// TIA Portal project "EB23" (V15)
// Maquina Raumak 23

(* hardware
DEVICE "S7-1200 station_1"  S7-1200 Station
   slot 0: "Rack_0"  S7-1200 Rack  Rack  V1.0
   slot 1: "PLC_1"  CPU 1214C DC/DC/Rly  6ES7 214-1HG40-0XB0  V4.2
   slot 2: "DI 16x24VDC_1"  6ES7 221-1BH32-0XB0  V2.0
   slot 3: "DQ 16x24VDC_1"  SM 1222 DQ16 x 24VDC  6ES7 222-1BH32-0XB0  V2.0
DEVICE "HMI_1"  KTP700 Basic PN
   slot 0: "HMI_1"  KTP700 Basic PN  6AV2 123-2GB03-0AX0  15.0.0.0
   slot 1: "HMI_RT_1"  KTP700 Basic PN  6AV2 123-2GB03-0AX0  15.0.0.0
   slot 5: "HMI_1.IE_CP_1"  PROFINET Interface  15.0.0.0
      slot 1: "PROFINET Interface_1"  PROFINET Interface
         slot 1: "Port_1"  Port
*)

// ===== PLC "PLC_1"  CPU 1214C DC/DC/Rly =====

VAR_GLOBAL   // PLC tag table "Default tag table"
   "System_Byte" AT %MB1 : Byte;
   "FirstScan" AT %M1.0 : Bool;
   "DiagStatusUpdate" AT %M1.1 : Bool;
   "AlwaysTRUE" AT %M1.2 : Bool;
   "AlwaysFALSE" AT %M1.3 : Bool;
   "Clock_Byte" AT %MB0 : Byte;
   "Clock_10Hz" AT %M0.0 : Bool;
   "Clock_5Hz" AT %M0.1 : Bool;
   "Clock_2.5Hz" AT %M0.2 : Bool;
   "Clock_2Hz" AT %M0.3 : Bool;
   "Clock_1.25Hz" AT %M0.4 : Bool;
   "Clock_1Hz" AT %M0.5 : Bool;
   "Clock_0.625Hz" AT %M0.6 : Bool;
   "Clock_0.5Hz" AT %M0.7 : Bool;
   "E_stop_bit" AT %M10.0 : Bool;
   "F_Blender_bit" AT %M10.1 : Bool;
   "F_Collector_bit" AT %M10.2 : Bool;
   "F_puller_bit" AT %M10.3 : Bool;
   "F_servo_bit" AT %M10.4 : Bool;
   "F_unwinder_bit" AT %M10.5 : Bool;
   "Global_Alarm" AT %M10.6 : Bool;
   "Doser_pulse" AT %I0.0 : Bool;   // HSC in
   "Stop" AT %I0.2 : Bool;   // Stops machine
   "Start" AT %I0.3 : Bool;   // Start machine
   "F_Collector" AT %I0.4 : Bool;   // Collector band termic fuse
   "S_Horizontalsealer" AT %I0.5 : Bool;   // Sensor Horizontal Sealer
   "S_Photocell" AT %I0.6 : Bool;   // Photocell sensor
   "F_Unwinder" AT %I0.7 : Bool;   // Unwinder Motor thermic fuse
   "S_Reedlvl" AT %I1.0 : Bool;   // level Switch
   "F_Servo" AT %I1.1 : Bool;   // Servo motor termic fuse
   "F_Puller" AT %I1.2 : Bool;   // Puller motor termic fuse
   "S_OpenDoor" AT %I1.3 : Bool;   // Sensor Action Open Door
   "F_Blender" AT %I1.4 : Bool;   // Blender Motor thermic fuse
   "E_stop" AT %I1.5 : Bool;   // Emergency Stop
   "S_StuckCoil" AT %I8.0 : Bool;   // Sensor Stuck coil
   "S_UnwinderOn" AT %I8.1 : Bool;   // Sensor unwinder On
   "S_UnwinderOff" AT %I8.2 : Bool;   // Sensor unwinder Off
   "S_LooseCoil" AT %I8.3 : Bool;   // Sensor Loose Coil
   "S_knife" AT %I8.4 : Bool;   // Sensor Knife
   "Stop_remote" AT %I8.5 : Bool;   // Stop Remote
   "Dater_fault" AT %I8.6 : Bool;   // Dater Fault (Print)
   "Coder" AT %Q0.0 : Bool;   // Out Coder EV
   "Horizontal_sealer" AT %Q0.1 : Bool;   // Out Horizontal Sealer EV
   "Vertical_sealer" AT %Q0.2 : Bool;   // Out Vertical Sealer EV
   "Knife" AT %Q0.3 : Bool;   // Out Knife EV
   "Puller" AT %Q0.4 : Bool;   // Out Drive Puller
   "Pusher" AT %Q0.5 : Bool;   // Out Pusher EV
   "HorizontalHeater" AT %Q0.6 : Bool;   // Out KS Horizontal Heater
   "VerticalHeater" AT %Q0.7 : Bool;   // Out KS Vertical Heater
   "Feeder" AT %Q1.0 : Bool;   // Out Feeder EV
   "Doser" AT %Q1.1 : Bool;   // Out Servo Drive Doser
   "Unwinder" AT %Q12.0 : Bool;   // Out Unwinder motor
   "CollectorBelt" AT %Q12.1 : Bool;   // Out Collector Belt motor
   "Blender" AT %Q12.2 : Bool;   // Out Blender motor
   "En_io_doser" AT %Q12.3 : Bool;   // Out Enable and Reset Servo Drive Doser
   "dater" AT %Q12.4 : Bool;   // Out dater(Print)
   "Doser_pulse_bit" AT %M10.7 : Bool;
   "Stop_bit" AT %M11.0 : Bool;
   "Start_bit" AT %M11.1 : Bool;
   "S_Horizontalsealer_bit" AT %M11.2 : Bool;
   "S_Photocell_bit" AT %M11.3 : Bool;
   "S_Reedlvl_bit" AT %M11.4 : Bool;
   "S_OpenDoor_bit" AT %M11.5 : Bool;
   "S_StuckCoil_bit" AT %M11.7 : Bool;
   "S_UnwinderOn_bit" AT %M12.0 : Bool;
   "S_UnwinderOff_bit" AT %M12.1 : Bool;
   "S_LooseCoil_bit" AT %M12.2 : Bool;
   "S_knife_bit" AT %M12.3 : Bool;
   "Stop_remote_bit" AT %M12.4 : Bool;
   "Dater_fault_bit" AT %M12.5 : Bool;
   "Coder_bit" AT %M12.6 : Bool;
   "Horizontal_sealer_bit" AT %M12.7 : Bool;
   "Vertical_sealer_bit" AT %M13.0 : Bool;
   "Knife_bit" AT %M13.1 : Bool;
   "Puller_bit" AT %M13.2 : Bool;
   "Pusher_bit" AT %M13.3 : Bool;
   "HorizontalHeater_bit" AT %M13.4 : Bool;
   "VerticalHeater_bit" AT %M13.5 : Bool;
   "Feeder_bit" AT %M13.6 : Bool;
   "Doser_bit" AT %M13.7 : Bool;
   "Unwinder_bit" AT %M14.0 : Bool;
   "CollectorBelt_bit" AT %M14.1 : Bool;
   "Blender_bit" AT %M14.2 : Bool;
   "En_io_doser_bit" AT %M14.3 : Bool;
   "dater_bit" AT %M14.4 : Bool;
   "ONS0" AT %M14.5 : Bool;
   "Stop_machine" AT %M14.6 : Bool;
   "Run" AT %M14.7 : Bool;
   "En_opendoor" AT %M15.0 : Bool;
   "Stop_1" AT %M15.1 : Bool;
   "Stop_2" AT %M15.2 : Bool;
   "Stop_3" AT %M15.3 : Bool;
   "Stop_4" AT %M15.4 : Bool;
   "Stop_5" AT %M15.5 : Bool;
   "Stop_6" AT %M15.6 : Bool;
   "En_conectionHMI" AT %M15.7 : Bool;
   "Stage_1" AT %M16.0 : Bool;   // Ingreso a Etapa
   "Stage_2" AT %M16.1 : Bool;   // Sellado EV Vertical
   "Stage_3" AT %M16.2 : Bool;   // Sellado EV Horizontal
   "Stage_4" AT %M16.3 : Bool;   // Dater Print
   "Stage_5" AT %M16.4 : Bool;   // Maquina armada... lista a Dispensar
   "Stage_6" AT %M16.5 : Bool;   // Etapa de Confirmacion de sellado
   "T_puller_run" AT %MD17 : Time;
   "Stage_0" AT %M16.6 : Bool;   // Etapa de Reinicio
   "E_Manual_hmi" AT %M16.7 : Bool;
   "E_Manual" AT %M21.0 : Bool;
   "En_Verticalsealer_hmi" AT %M21.1 : Bool;
   "TestVerticalsealer_hmi" AT %M21.2 : Bool;
   "En_Horizontalsealer_hmi" AT %M21.3 : Bool;
   "Testhorizontalsealer_hmi" AT %M21.4 : Bool;
   "En_dater_hmi" AT %M21.5 : Bool;
   "Testdater_hmi" AT %M21.6 : Bool;
   "En_doser_hmi" AT %M21.7 : Bool;
   "En_knife_hmi" AT %M22.0 : Bool;
   "Tag_2" AT %M22.1 : Bool;
   "TestKnife_hmi" AT %M22.2 : Bool;
   "Stage_7" AT %M22.3 : Bool;   // Dosificar
   "Stage_8" AT %M22.4 : Bool;   // Corte cuchillo Ristra
   "Stage_9_1" AT %M22.5 : Bool;
   "ONS2" AT %M22.6 : Bool;
   "Testdoser_hmi" AT %M22.7 : Bool;
   "Stage_9_2" AT %M23.0 : Bool;
   "En_colector_hmi" AT %M23.1 : Bool;
   "TestCollector_hmi" AT %M23.2 : Bool;
   "En_Feeder_hmi" AT %M23.3 : Bool;
   "Stage_Feed_1" AT %M23.4 : Bool;
   "Stage_Blender_1" AT %M23.5 : Bool;
   "TestFeeder_hmi" AT %M23.6 : Bool;
   "En_blender_hmi" AT %M23.7 : Bool;
   "TestBlender_hmi" AT %M24.0 : Bool;
   "En_pusher_hmi" AT %M24.1 : Bool;
   "En_cleaning_hmi" AT %M24.2 : Bool;
   "Stage_CleaningMachine" AT %M24.3 : Bool;
   "Stage_Pusher" AT %M24.4 : Bool;
   "TestPusher_hmi" AT %M24.5 : Bool;
   "En_horizontalheater_hmi" AT %M24.6 : Bool;
   "En_verticalheater_hmi" AT %M24.7 : Bool;
   "Stage_9_0" AT %M25.0 : Bool;
   "Stage_Feed_0" AT %M25.1 : Bool;
   "Stage_Unw_0" AT %M25.2 : Bool;
   "Stage_Unw_1" AT %M25.3 : Bool;
   "En_puller_hmi" AT %M25.4 : Bool;
   "ONS5" AT %M25.5 : Bool;
   "TestUnwinder_hmi" AT %M25.6 : Bool;
   "Stage_Puller_1" AT %M25.7 : Bool;
   "Tag_3" AT %M26.0 : Bool;
   "Et_puller" AT %MD27 : Time;
   "U_Coder_bit" AT %M31.0 : Bool;
   "TestPuller_hmi" AT %M31.1 : Bool;
   "Stage_Photo_1" AT %M31.2 : Bool;
   "ONS7" AT %M31.3 : Bool;
   "Stage_Photo_0" AT %M31.4 : Bool;
   "ONS8" AT %M31.5 : Bool;
   "reset_ppm" AT %M31.6 : Bool;
   "CV_ppm" AT %MW32 : Int;
   "ONS10" AT %M34.0 : Bool;
   "PPM" AT %MW36 : Int;
   "Total_vertical_sealer" AT %MD38 : Time;
   "High_Sealer" AT %MD42 : Time;
   "stimate_ppm" AT %MD46 : DInt;
   "ret_val_RD_LOC" AT %MW50 : Int;
   "ret_val_RD_SYS" AT %MW52 : Int;
   "ret_val_WR_SYS" AT %MW54 : Int;
   "ONS12" AT %M56.0 : Bool;
   "write_time" AT %M56.1 : Bool;
   "Stage_Blender_0" AT %M56.2 : Bool;
END_VAR

DATA_BLOCK "DB_Alarms"   // DB1
{ S7_Optimized_Access := 'FALSE' }
VERSION : 0.1
   VAR
      Alarms_active : Bool;
      E_stop_alm : Bool;
      Colector_alm : Bool;
      Puller_alm : Bool;
      "Unwinder-alm" : Bool;
      Servo_alm : Bool;
      Blender_alm : Bool;
      Open_door : Bool;
      Remote_stop : Bool;
      No_product : Bool;
      Blocked_jaws : Bool;
      Unwinder_loose : Bool;
      Unwinder_stuck : Bool;
      Stop_photocell : Bool;
      Coder_alm : Bool;
      Feed_alm : Bool;
   END_VAR
BEGIN
END_DATA_BLOCK

DATA_BLOCK "Init_Var"   // DB2
{ S7_Optimized_Access := 'TRUE' }
VERSION : 0.1
   VAR RETAIN
      Pt_cleaning : Time;
      Pt_coder : Time;
      Pt_collector : Time;
      Pt_collector_cut : Time;
      Pt_delay_doser : Time;
      Pt_delay_vert : Time;
      Pt_feeder : Time;
      Pt_horizontalsealer : Time;
      Pt_knife : Time;
      Pt_photocell : Time;
      Pt_preheat : Time;
      Pt_Puller : Time;
      Pt_pulses : Time;
      Pt_verticalsealer : Time;
      N_cycles : Int;
   END_VAR
BEGIN
END_DATA_BLOCK

DATA_BLOCK "DB_Time"   // DB22
{ S7_Optimized_Access := 'TRUE' }
VERSION : 0.1
   VAR
      time_local_READ : DTL;
      time_system_READ : DTL;
      time_system_WRITE : DTL;
   END_VAR
BEGIN
END_DATA_BLOCK

DATA_BLOCK "db_time_sync"   // DB22
{ S7_Optimized_Access := 'TRUE' }
VERSION : 0.1
   VAR
      time_local_READ : DTL;
      time_system_READ : DTL;
      time_system_WRITE : DTL;
   END_VAR
BEGIN
END_DATA_BLOCK

// folder: System blocks/Program resources

DATA_BLOCK "T_horizontal_stop"   // DB3
{ S7_Optimized_Access := 'TRUE' }
AUTHOR : Simatic
FAMILY : IEC
NAME : IEC_TMR
VERSION : 1.0
// stored: InstanceOfName IEC_TIMER
"IEC_TIMER"
BEGIN
END_DATA_BLOCK

DATA_BLOCK "T_delay_vert"   // DB4
{ S7_Optimized_Access := 'TRUE' }
AUTHOR : Simatic
FAMILY : IEC
NAME : IEC_TMR
VERSION : 1.0
// stored: InstanceOfName IEC_TIMER
"IEC_TIMER"
BEGIN
END_DATA_BLOCK

DATA_BLOCK "T_VerticalS"   // DB5
{ S7_Optimized_Access := 'TRUE' }
AUTHOR : Simatic
FAMILY : IEC
NAME : IEC_TMR
VERSION : 1.0
// stored: InstanceOfName IEC_TIMER
"IEC_TIMER"
BEGIN
END_DATA_BLOCK

DATA_BLOCK "T_HorizontalSealer"   // DB6
{ S7_Optimized_Access := 'TRUE' }
AUTHOR : Simatic
FAMILY : IEC
NAME : IEC_TMR
VERSION : 1.0
// stored: InstanceOfName IEC_TIMER
"IEC_TIMER"
BEGIN
END_DATA_BLOCK

DATA_BLOCK "Packages_Knife"   // DB7
{ S7_Optimized_Access := 'TRUE' }
AUTHOR : Simatic
FAMILY : IEC
NAME : CNTR
VERSION : 1.0
// stored: InstanceOfName IEC_COUNTER
"IEC_COUNTER"
BEGIN
END_DATA_BLOCK

DATA_BLOCK "T_Knife"   // DB8
{ S7_Optimized_Access := 'TRUE' }
AUTHOR : Simatic
FAMILY : IEC
NAME : IEC_TMR
VERSION : 1.0
// stored: InstanceOfName IEC_TIMER
"IEC_TIMER"
BEGIN
END_DATA_BLOCK

DATA_BLOCK "T_DelayDoser"   // DB9
{ S7_Optimized_Access := 'TRUE' }
AUTHOR : Simatic
FAMILY : IEC
NAME : IEC_TMR
VERSION : 1.0
// stored: InstanceOfName IEC_TIMER
"IEC_TIMER"
BEGIN
END_DATA_BLOCK

DATA_BLOCK "T_PulseDoser"   // DB10
{ S7_Optimized_Access := 'TRUE' }
AUTHOR : Simatic
FAMILY : IEC
NAME : IEC_TMR
VERSION : 1.0
// stored: InstanceOfName IEC_TIMER
"IEC_TIMER"
BEGIN
END_DATA_BLOCK

DATA_BLOCK "T_CollectorCut"   // DB11
{ S7_Optimized_Access := 'TRUE' }
AUTHOR : Simatic
FAMILY : IEC
NAME : IEC_TMR
VERSION : 1.0
// stored: InstanceOfName IEC_TIMER
"IEC_TIMER"
BEGIN
END_DATA_BLOCK

DATA_BLOCK "T_Collector"   // DB12
{ S7_Optimized_Access := 'TRUE' }
AUTHOR : Simatic
FAMILY : IEC
NAME : IEC_TMR
VERSION : 1.0
// stored: InstanceOfName IEC_TIMER
"IEC_TIMER"
BEGIN
END_DATA_BLOCK

DATA_BLOCK "Cnt_LevelFeeder"   // DB13
{ S7_Optimized_Access := 'TRUE' }
AUTHOR : Simatic
FAMILY : IEC
NAME : CNTR
VERSION : 1.0
// stored: InstanceOfName IEC_COUNTER
"IEC_COUNTER"
BEGIN
END_DATA_BLOCK

DATA_BLOCK "T_Feeder"   // DB14
{ S7_Optimized_Access := 'TRUE' }
AUTHOR : Simatic
FAMILY : IEC
NAME : IEC_TMR
VERSION : 1.0
// stored: InstanceOfName IEC_TIMER
"IEC_TIMER"
BEGIN
END_DATA_BLOCK

DATA_BLOCK "T_CleanMachine"   // DB15
{ S7_Optimized_Access := 'TRUE' }
AUTHOR : Simatic
FAMILY : IEC
NAME : IEC_TMR
VERSION : 1.0
// stored: InstanceOfName IEC_TIMER
"IEC_TIMER"
BEGIN
END_DATA_BLOCK

DATA_BLOCK "T_Puller"   // DB16
{ S7_Optimized_Access := 'TRUE' }
AUTHOR : Simatic
FAMILY : IEC
NAME : IEC_TMR
VERSION : 1.0
// stored: InstanceOfName IEC_TIMER
"IEC_TIMER"
BEGIN
END_DATA_BLOCK

DATA_BLOCK "T_Puller_Running"   // DB17
{ S7_Optimized_Access := 'TRUE' }
AUTHOR : Simatic
FAMILY : IEC
NAME : IEC_TMR
VERSION : 1.0
// stored: InstanceOfName IEC_TIMER
"IEC_TIMER"
BEGIN
END_DATA_BLOCK

DATA_BLOCK "T_PhotoCell"   // DB18
{ S7_Optimized_Access := 'TRUE' }
AUTHOR : Simatic
FAMILY : IEC
NAME : IEC_TMR
VERSION : 1.0
// stored: InstanceOfName IEC_TIMER
"IEC_TIMER"
BEGIN
END_DATA_BLOCK

DATA_BLOCK "Packages_PPM"   // DB19
{ S7_Optimized_Access := 'TRUE' }
AUTHOR : Simatic
FAMILY : IEC
NAME : CNTR
VERSION : 1.0
// stored: InstanceOfName IEC_COUNTER
"IEC_COUNTER"
BEGIN
END_DATA_BLOCK

DATA_BLOCK "T_Delay_ppm"   // DB20
{ S7_Optimized_Access := 'TRUE' }
AUTHOR : Simatic
FAMILY : IEC
NAME : IEC_TMR
VERSION : 1.0
// stored: InstanceOfName IEC_TIMER
"IEC_TIMER"
BEGIN
END_DATA_BLOCK

DATA_BLOCK "T_ppm"   // DB21
{ S7_Optimized_Access := 'TRUE' }
AUTHOR : Simatic
FAMILY : IEC
NAME : IEC_TMR
VERSION : 1.0
// stored: InstanceOfName IEC_TIMER
"IEC_TIMER"
BEGIN
END_DATA_BLOCK

// folder: (top level)

ORGANIZATION_BLOCK "Main"   // OB1, LAD, ProgramCycle
TITLE = "Main Program Sweep (Cycle)"
{ S7_Optimized_Access := 'TRUE' }
VERSION : 0.1
   VAR_INPUT
      Initial_Call : Bool;   // Initial call of this OB
      Remanence : Bool;   // =True, if remanent data are available
   END_VAR
   VAR_TEMP   // added for the SCL form of the ladder/FBD networks
      _w1 : Bool;
   END_VAR
BEGIN

REGION Network 1
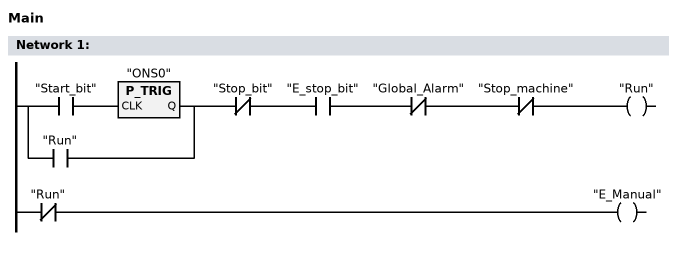
   RUNG wire#powerrail
      Contact( "Start_bit" )
      P_Trig( "ONS0" )
      wire#w1
      I_Contact( "Stop_bit" )
      Contact( "E_stop_bit" )
      I_Contact( "Global_Alarm" )
      I_Contact( "Stop_machine" )
      Coil( "Run" )
   END_RUNG
   RUNG wire#powerrail
      Contact( "Run" )
   END_RUNG wire#w1
   RUNG wire#powerrail
      I_Contact( "Run" )
      Coil( "E_Manual" )
   END_RUNG
   // the same network as SCL:
   #_w1 := "Start_bit" AND NOT "ONS0";   // rising edge
   "ONS0" := "Start_bit";
   "Run" := (#_w1 OR "Run") AND NOT "Stop_bit" AND "E_stop_bit" AND NOT "Global_Alarm" AND NOT "Stop_machine";
   "E_Manual" := NOT "Run";
END_REGION
END_ORGANIZATION_BLOCK

ORGANIZATION_BLOCK "Actions"   // OB123, LAD, ProgramCycle
TITLE = "Main Program Sweep (Cycle)"
{ S7_Optimized_Access := 'TRUE' }
VERSION : 0.1
   VAR_INPUT
      Initial_Call : Bool;   // Initial call of this OB
      Remanence : Bool;   // =True, if remanent data are available
   END_VAR
BEGIN

REGION Network 1: Peripherals EV
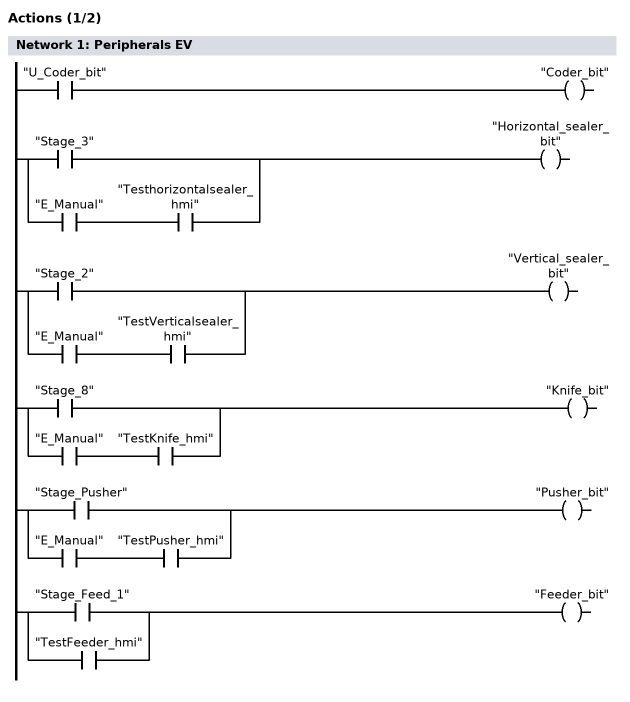
   RUNG wire#powerrail
      Contact( "U_Coder_bit" )
      Coil( "Coder_bit" )
   END_RUNG
   RUNG wire#powerrail
      Contact( "Stage_3" )
      wire#w1
      Coil( "Horizontal_sealer_bit" )
   END_RUNG
   RUNG wire#powerrail
      Contact( "E_Manual" )
      Contact( "Testhorizontalsealer_hmi" )
   END_RUNG wire#w1
   RUNG wire#powerrail
      Contact( "Stage_2" )
      wire#w2
      Coil( "Vertical_sealer_bit" )
   END_RUNG
   RUNG wire#powerrail
      Contact( "E_Manual" )
      Contact( "TestVerticalsealer_hmi" )
   END_RUNG wire#w2
   RUNG wire#powerrail
      Contact( "Stage_8" )
      wire#w3
      Coil( "Knife_bit" )
   END_RUNG
   RUNG wire#powerrail
      Contact( "E_Manual" )
      Contact( "TestKnife_hmi" )
   END_RUNG wire#w3
   RUNG wire#powerrail
      Contact( "Stage_Pusher" )
      wire#w4
      Coil( "Pusher_bit" )
   END_RUNG
   RUNG wire#powerrail
      Contact( "E_Manual" )
      Contact( "TestPusher_hmi" )
   END_RUNG wire#w4
   RUNG wire#powerrail
      Contact( "Stage_Feed_1" )
      wire#w5
      Coil( "Feeder_bit" )
   END_RUNG
   RUNG wire#powerrail
      Contact( "TestFeeder_hmi" )
   END_RUNG wire#w5
   // the same network as SCL:
   "Coder_bit" := "U_Coder_bit";
   "Horizontal_sealer_bit" := "Stage_3" OR ("E_Manual" AND "Testhorizontalsealer_hmi");
   "Vertical_sealer_bit" := "Stage_2" OR ("E_Manual" AND "TestVerticalsealer_hmi");
   "Knife_bit" := "Stage_8" OR ("E_Manual" AND "TestKnife_hmi");
   "Pusher_bit" := "Stage_Pusher" OR ("E_Manual" AND "TestPusher_hmi");
   "Feeder_bit" := "Stage_Feed_1" OR "TestFeeder_hmi";
END_REGION

REGION Network 2: Peripherals Motors
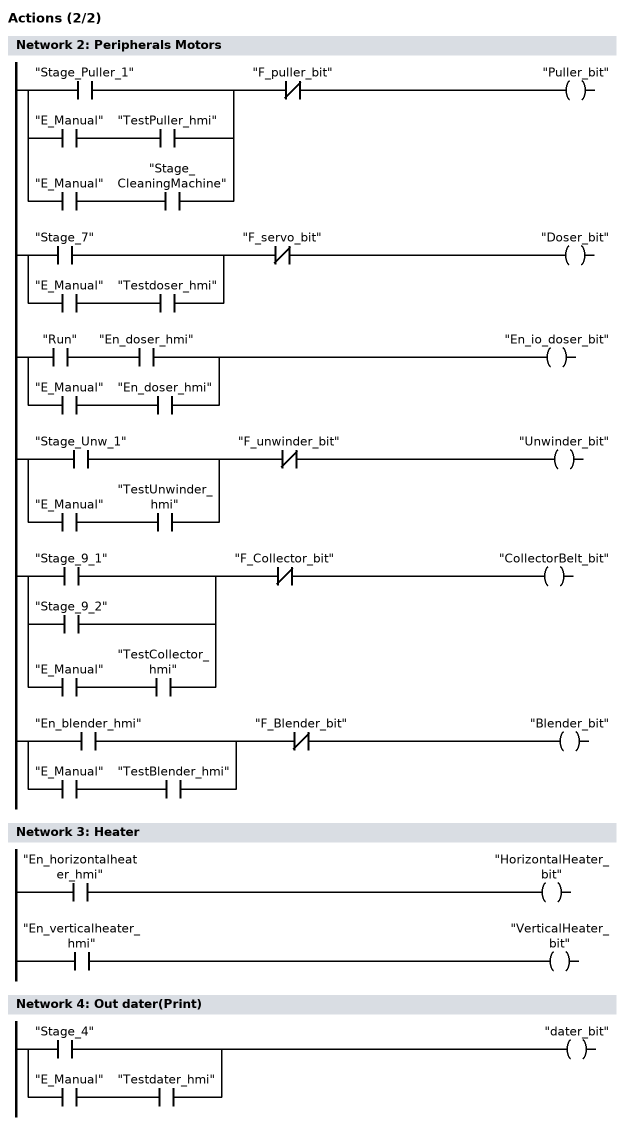
   RUNG wire#powerrail
      Contact( "Stage_Puller_1" )
      wire#w1
      I_Contact( "F_puller_bit" )
      Coil( "Puller_bit" )
   END_RUNG
   RUNG wire#powerrail
      Contact( "E_Manual" )
      Contact( "TestPuller_hmi" )
   END_RUNG wire#w1
   RUNG wire#powerrail
      Contact( "E_Manual" )
      Contact( "Stage_CleaningMachine" )
   END_RUNG wire#w1
   RUNG wire#powerrail
      Contact( "Stage_7" )
      wire#w2
      I_Contact( "F_servo_bit" )
      Coil( "Doser_bit" )
   END_RUNG
   RUNG wire#powerrail
      Contact( "E_Manual" )
      Contact( "Testdoser_hmi" )
   END_RUNG wire#w2
   RUNG wire#powerrail
      Contact( "Run" )
      Contact( "En_doser_hmi" )
      wire#w3
      Coil( "En_io_doser_bit" )
   END_RUNG
   RUNG wire#powerrail
      Contact( "E_Manual" )
      Contact( "En_doser_hmi" )
   END_RUNG wire#w3
   RUNG wire#powerrail
      Contact( "Stage_Unw_1" )
      wire#w4
      I_Contact( "F_unwinder_bit" )
      Coil( "Unwinder_bit" )
   END_RUNG
   RUNG wire#powerrail
      Contact( "E_Manual" )
      Contact( "TestUnwinder_hmi" )
   END_RUNG wire#w4
   RUNG wire#powerrail
      Contact( "Stage_9_1" )
      wire#w5
      I_Contact( "F_Collector_bit" )
      Coil( "CollectorBelt_bit" )
   END_RUNG
   RUNG wire#powerrail
      Contact( "Stage_9_2" )
   END_RUNG wire#w5
   RUNG wire#powerrail
      Contact( "E_Manual" )
      Contact( "TestCollector_hmi" )
   END_RUNG wire#w5
   RUNG wire#powerrail
      Contact( "En_blender_hmi" )
      wire#w6
      I_Contact( "F_Blender_bit" )
      Coil( "Blender_bit" )
   END_RUNG
   RUNG wire#powerrail
      Contact( "E_Manual" )
      Contact( "TestBlender_hmi" )
   END_RUNG wire#w6
   // the same network as SCL:
   "Puller_bit" := ("Stage_Puller_1" OR ("E_Manual" AND "TestPuller_hmi") OR ("E_Manual" AND "Stage_CleaningMachine")) AND NOT "F_puller_bit";
   "Doser_bit" := ("Stage_7" OR ("E_Manual" AND "Testdoser_hmi")) AND NOT "F_servo_bit";
   "En_io_doser_bit" := ("Run" AND "En_doser_hmi") OR ("E_Manual" AND "En_doser_hmi");
   "Unwinder_bit" := ("Stage_Unw_1" OR ("E_Manual" AND "TestUnwinder_hmi")) AND NOT "F_unwinder_bit";
   "CollectorBelt_bit" := ("Stage_9_1" OR "Stage_9_2" OR ("E_Manual" AND "TestCollector_hmi")) AND NOT "F_Collector_bit";
   "Blender_bit" := ("En_blender_hmi" OR ("E_Manual" AND "TestBlender_hmi")) AND NOT "F_Blender_bit";
END_REGION

REGION Network 3: Heater
   RUNG wire#powerrail
      Contact( "En_horizontalheater_hmi" )
      Coil( "HorizontalHeater_bit" )
   END_RUNG
   RUNG wire#powerrail
      Contact( "En_verticalheater_hmi" )
      Coil( "VerticalHeater_bit" )
   END_RUNG
   // the same network as SCL:
   "HorizontalHeater_bit" := "En_horizontalheater_hmi";
   "VerticalHeater_bit" := "En_verticalheater_hmi";
END_REGION

REGION Network 4: Out dater(Print)
   RUNG wire#powerrail
      Contact( "Stage_4" )
      wire#w1
      Coil( "dater_bit" )
   END_RUNG
   RUNG wire#powerrail
      Contact( "E_Manual" )
      Contact( "Testdater_hmi" )
   END_RUNG wire#w1
   // the same network as SCL:
   "dater_bit" := "Stage_4" OR ("E_Manual" AND "Testdater_hmi");
END_REGION
END_ORGANIZATION_BLOCK

ORGANIZATION_BLOCK "Alarms"   // OB124, LAD, ProgramCycle
TITLE = "Main Program Sweep (Cycle)"
{ S7_Optimized_Access := 'TRUE' }
VERSION : 0.1
   VAR_INPUT
      Initial_Call : Bool;   // Initial call of this OB
      Remanence : Bool;   // =True, if remanent data are available
   END_VAR
BEGIN

REGION Network 1: Global Alarm Fuses
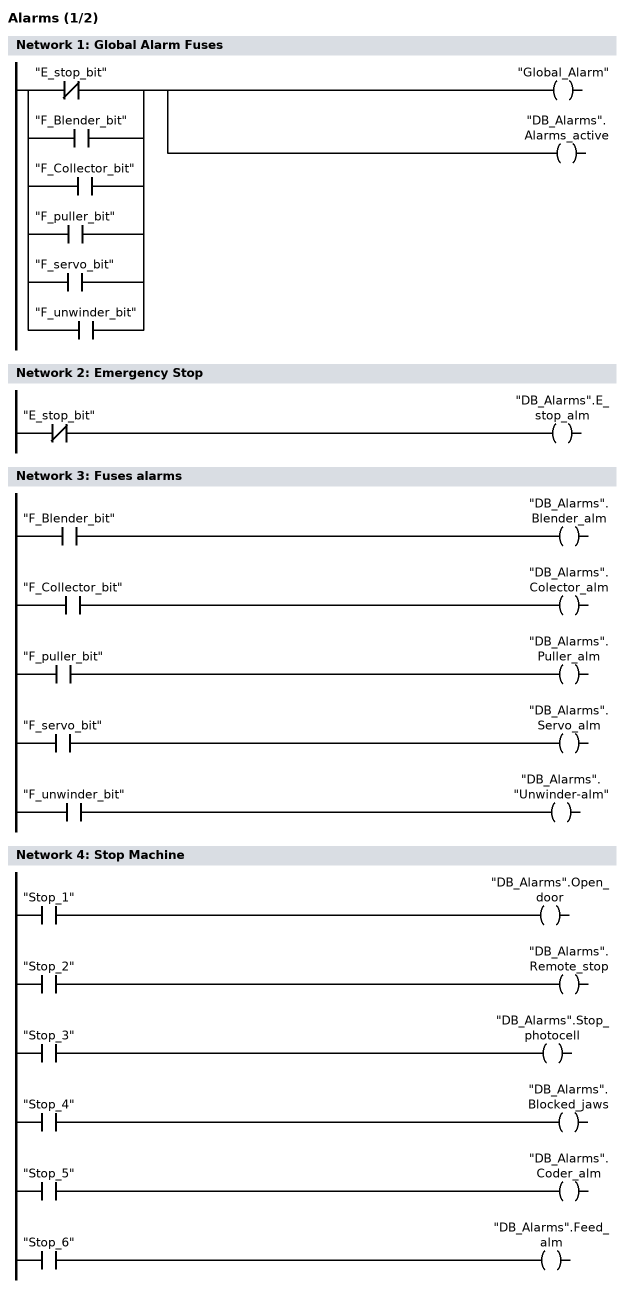
   RUNG wire#powerrail
      I_Contact( "E_stop_bit" )
      wire#w1
      Coil( "Global_Alarm" )
   END_RUNG
   RUNG wire#powerrail
      Contact( "F_Blender_bit" )
   END_RUNG wire#w1
   RUNG wire#powerrail
      Contact( "F_Collector_bit" )
   END_RUNG wire#w1
   RUNG wire#powerrail
      Contact( "F_puller_bit" )
   END_RUNG wire#w1
   RUNG wire#powerrail
      Contact( "F_servo_bit" )
   END_RUNG wire#w1
   RUNG wire#powerrail
      Contact( "F_unwinder_bit" )
   END_RUNG wire#w1
   RUNG wire#w1
      Coil( "DB_Alarms".Alarms_active )
   END_RUNG
   // the same network as SCL:
   "Global_Alarm" := NOT "E_stop_bit" OR "F_Blender_bit" OR "F_Collector_bit" OR "F_puller_bit" OR "F_servo_bit" OR "F_unwinder_bit";
   "DB_Alarms".Alarms_active := "Global_Alarm";
END_REGION

REGION Network 2: Emergency Stop
   RUNG wire#powerrail
      I_Contact( "E_stop_bit" )
      Coil( "DB_Alarms".E_stop_alm )
   END_RUNG
   // the same network as SCL:
   "DB_Alarms".E_stop_alm := NOT "E_stop_bit";
END_REGION

REGION Network 3: Fuses alarms
   RUNG wire#powerrail
      Contact( "F_Blender_bit" )
      Coil( "DB_Alarms".Blender_alm )
   END_RUNG
   RUNG wire#powerrail
      Contact( "F_Collector_bit" )
      Coil( "DB_Alarms".Colector_alm )
   END_RUNG
   RUNG wire#powerrail
      Contact( "F_puller_bit" )
      Coil( "DB_Alarms".Puller_alm )
   END_RUNG
   RUNG wire#powerrail
      Contact( "F_servo_bit" )
      Coil( "DB_Alarms".Servo_alm )
   END_RUNG
   RUNG wire#powerrail
      Contact( "F_unwinder_bit" )
      Coil( "DB_Alarms"."Unwinder-alm" )
   END_RUNG
   // the same network as SCL:
   "DB_Alarms".Blender_alm := "F_Blender_bit";
   "DB_Alarms".Colector_alm := "F_Collector_bit";
   "DB_Alarms".Puller_alm := "F_puller_bit";
   "DB_Alarms".Servo_alm := "F_servo_bit";
   "DB_Alarms"."Unwinder-alm" := "F_unwinder_bit";
END_REGION

REGION Network 4: Stop Machine
   RUNG wire#powerrail
      Contact( "Stop_1" )
      Coil( "DB_Alarms".Open_door )
   END_RUNG
   RUNG wire#powerrail
      Contact( "Stop_2" )
      Coil( "DB_Alarms".Remote_stop )
   END_RUNG
   RUNG wire#powerrail
      Contact( "Stop_3" )
      Coil( "DB_Alarms".Stop_photocell )
   END_RUNG
   RUNG wire#powerrail
      Contact( "Stop_4" )
      Coil( "DB_Alarms".Blocked_jaws )
   END_RUNG
   RUNG wire#powerrail
      Contact( "Stop_5" )
      Coil( "DB_Alarms".Coder_alm )
   END_RUNG
   RUNG wire#powerrail
      Contact( "Stop_6" )
      Coil( "DB_Alarms".Feed_alm )
   END_RUNG
   // the same network as SCL:
   "DB_Alarms".Open_door := "Stop_1";
   "DB_Alarms".Remote_stop := "Stop_2";
   "DB_Alarms".Stop_photocell := "Stop_3";
   "DB_Alarms".Blocked_jaws := "Stop_4";
   "DB_Alarms".Coder_alm := "Stop_5";
   "DB_Alarms".Feed_alm := "Stop_6";
END_REGION

REGION Network 5: Sensor Alarms
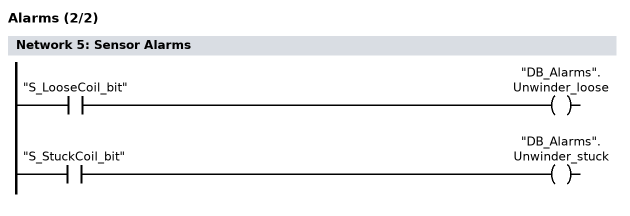
   RUNG wire#powerrail
      Contact( "S_LooseCoil_bit" )
      Coil( "DB_Alarms".Unwinder_loose )
   END_RUNG
   RUNG wire#powerrail
      Contact( "S_StuckCoil_bit" )
      Coil( "DB_Alarms".Unwinder_stuck )
   END_RUNG
   // the same network as SCL:
   "DB_Alarms".Unwinder_loose := "S_LooseCoil_bit";
   "DB_Alarms".Unwinder_stuck := "S_StuckCoil_bit";
END_REGION
END_ORGANIZATION_BLOCK

ORGANIZATION_BLOCK "Convertions"   // OB125, LAD, ProgramCycle
TITLE = "Main Program Sweep (Cycle)"
{ S7_Optimized_Access := 'TRUE' }
VERSION : 0.1
   VAR_INPUT
      Initial_Call : Bool;   // Initial call of this OB
      Remanence : Bool;   // =True, if remanent data are available
   END_VAR
   VAR_TEMP   // added for the SCL form of the ladder/FBD networks
      _w1 : Bool;
      _w2 : Bool;
      _w3 : Bool;
   END_VAR
BEGIN

REGION Network 2
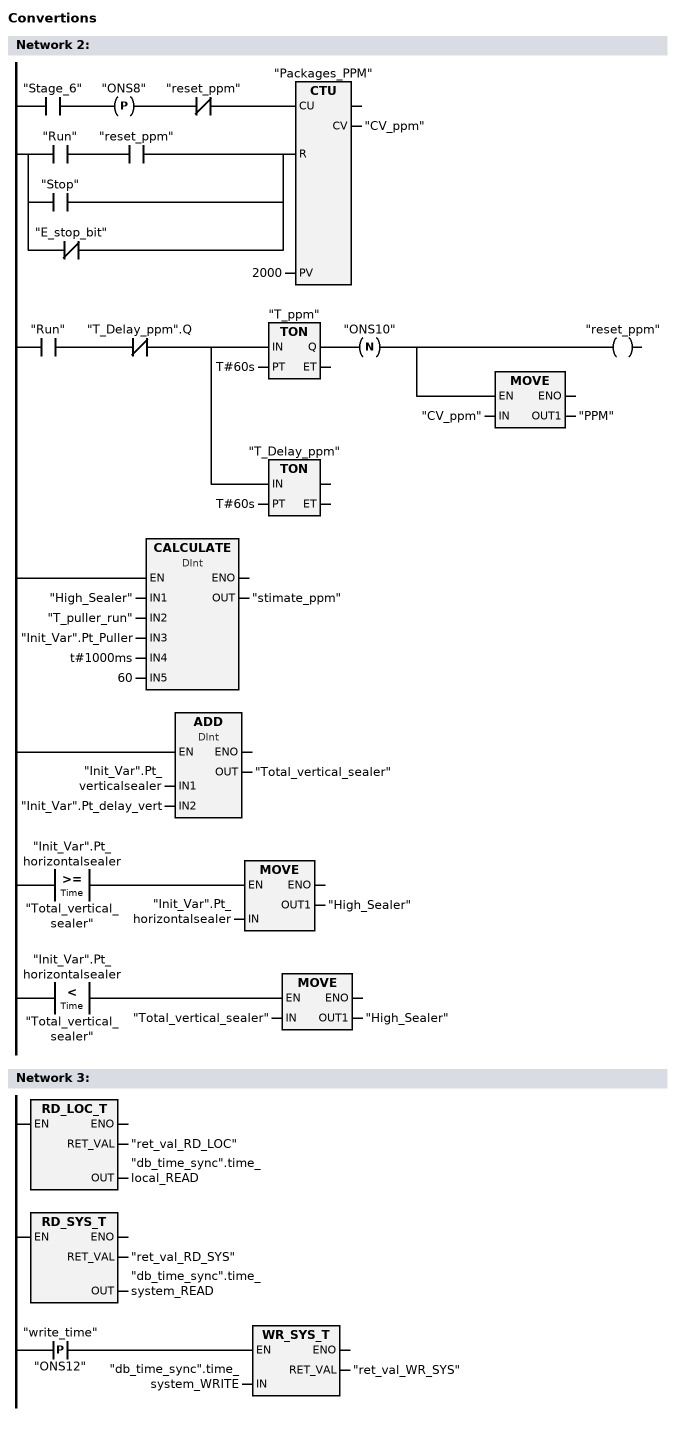
   #_w1 := "Stage_6" AND NOT "ONS8";   // rising edge
   "ONS8" := "Stage_6";
   "Packages_PPM".CTU(CU := #_w1 AND NOT "reset_ppm",
                      R := ("Run" AND "reset_ppm") OR "Stop" OR NOT "E_stop_bit",
                      PV := 2000,
                      CV => "CV_ppm");
   #_w2 := "Run" AND NOT "T_Delay_ppm".Q;
   "T_ppm".TON(IN := #_w2, PT := T#60s);
   #_w3 := NOT "T_ppm".Q AND "ONS10";   // falling edge
   "ONS10" := "T_ppm".Q;
   "reset_ppm" := #_w3;
   IF #_w3 THEN "PPM" := "CV_ppm"; END_IF;
   "T_Delay_ppm".TON(IN := #_w2, PT := T#60s);
   "stimate_ppm" := (t#1000ms*60)/("High_Sealer"+"T_puller_run"+"Init_Var".Pt_Puller);
   "Total_vertical_sealer" := "Init_Var".Pt_verticalsealer + "Init_Var".Pt_delay_vert;
   IF "Init_Var".Pt_horizontalsealer >= "Total_vertical_sealer" THEN
       "High_Sealer" := "Init_Var".Pt_horizontalsealer;
   END_IF;
   IF "Init_Var".Pt_horizontalsealer < "Total_vertical_sealer" THEN
       "High_Sealer" := "Total_vertical_sealer";
   END_IF;
END_REGION

REGION Network 3
   "ret_val_RD_LOC" := RD_LOC_T(OUT => "db_time_sync".time_local_READ);
   "ret_val_RD_SYS" := RD_SYS_T(OUT => "db_time_sync".time_system_READ);
   #_w1 := "write_time" AND NOT "ONS12";   // rising edge of "write_time"
   "ONS12" := "write_time";
   IF #_w1 THEN "ret_val_WR_SYS" := WR_SYS_T(IN := "db_time_sync".time_system_WRITE); END_IF;
END_REGION
END_ORGANIZATION_BLOCK

ORGANIZATION_BLOCK "Mirror_bit"   // OB126, LAD, ProgramCycle
TITLE = "Main Program Sweep (Cycle)"
{ S7_Optimized_Access := 'TRUE' }
VERSION : 0.1
   VAR_INPUT
      Initial_Call : Bool;   // Initial call of this OB
      Remanence : Bool;   // =True, if remanent data are available
   END_VAR
BEGIN

REGION Network 1: Inputs mirros Emergency
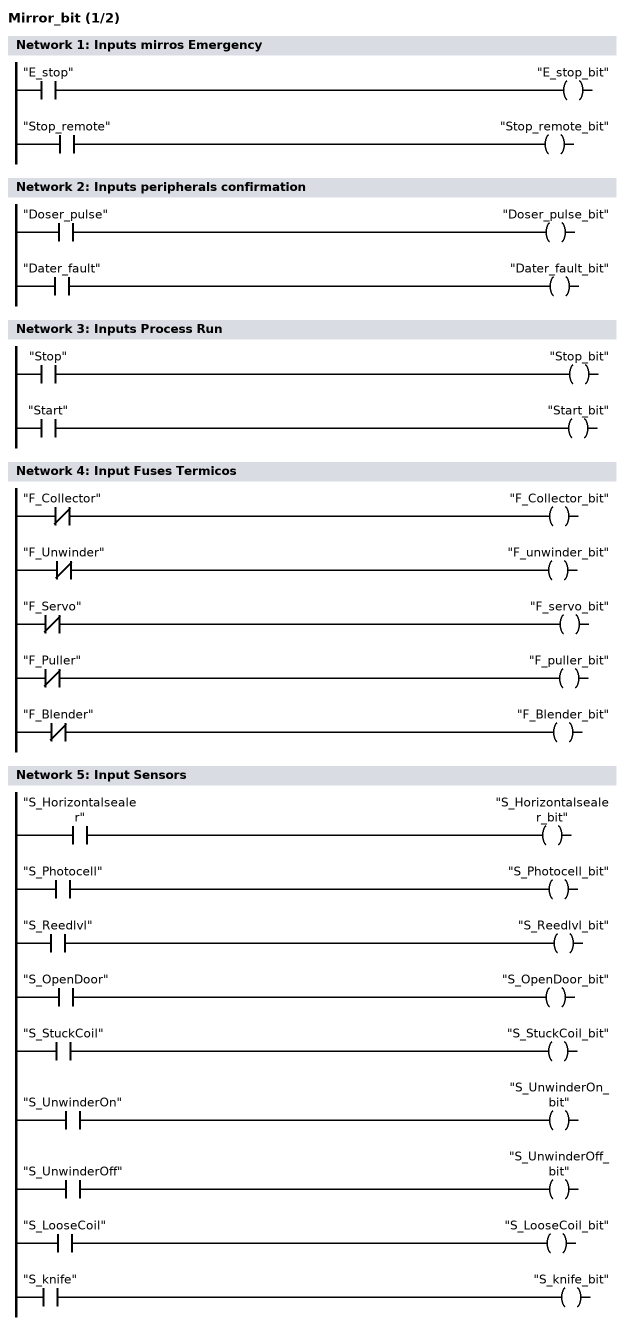
   RUNG wire#powerrail
      Contact( "E_stop" )
      Coil( "E_stop_bit" )
   END_RUNG
   RUNG wire#powerrail
      Contact( "Stop_remote" )
      Coil( "Stop_remote_bit" )
   END_RUNG
   // the same network as SCL:
   "E_stop_bit" := "E_stop";
   "Stop_remote_bit" := "Stop_remote";
END_REGION

REGION Network 2: Inputs peripherals confirmation
   RUNG wire#powerrail
      Contact( "Doser_pulse" )
      Coil( "Doser_pulse_bit" )
   END_RUNG
   RUNG wire#powerrail
      Contact( "Dater_fault" )
      Coil( "Dater_fault_bit" )
   END_RUNG
   // the same network as SCL:
   "Doser_pulse_bit" := "Doser_pulse";
   "Dater_fault_bit" := "Dater_fault";
END_REGION

REGION Network 3: Inputs Process Run
   RUNG wire#powerrail
      Contact( "Stop" )
      Coil( "Stop_bit" )
   END_RUNG
   RUNG wire#powerrail
      Contact( "Start" )
      Coil( "Start_bit" )
   END_RUNG
   // the same network as SCL:
   "Stop_bit" := "Stop";
   "Start_bit" := "Start";
END_REGION

REGION Network 4: Input Fuses Termicos
   RUNG wire#powerrail
      I_Contact( "F_Collector" )
      Coil( "F_Collector_bit" )
   END_RUNG
   RUNG wire#powerrail
      I_Contact( "F_Unwinder" )
      Coil( "F_unwinder_bit" )
   END_RUNG
   RUNG wire#powerrail
      I_Contact( "F_Servo" )
      Coil( "F_servo_bit" )
   END_RUNG
   RUNG wire#powerrail
      I_Contact( "F_Puller" )
      Coil( "F_puller_bit" )
   END_RUNG
   RUNG wire#powerrail
      I_Contact( "F_Blender" )
      Coil( "F_Blender_bit" )
   END_RUNG
   // the same network as SCL:
   "F_Collector_bit" := NOT "F_Collector";
   "F_unwinder_bit" := NOT "F_Unwinder";
   "F_servo_bit" := NOT "F_Servo";
   "F_puller_bit" := NOT "F_Puller";
   "F_Blender_bit" := NOT "F_Blender";
END_REGION

REGION Network 5: Input Sensors
   RUNG wire#powerrail
      Contact( "S_Horizontalsealer" )
      Coil( "S_Horizontalsealer_bit" )
   END_RUNG
   RUNG wire#powerrail
      Contact( "S_Photocell" )
      Coil( "S_Photocell_bit" )
   END_RUNG
   RUNG wire#powerrail
      Contact( "S_Reedlvl" )
      Coil( "S_Reedlvl_bit" )
   END_RUNG
   RUNG wire#powerrail
      Contact( "S_OpenDoor" )
      Coil( "S_OpenDoor_bit" )
   END_RUNG
   RUNG wire#powerrail
      Contact( "S_StuckCoil" )
      Coil( "S_StuckCoil_bit" )
   END_RUNG
   RUNG wire#powerrail
      Contact( "S_UnwinderOn" )
      Coil( "S_UnwinderOn_bit" )
   END_RUNG
   RUNG wire#powerrail
      Contact( "S_UnwinderOff" )
      Coil( "S_UnwinderOff_bit" )
   END_RUNG
   RUNG wire#powerrail
      Contact( "S_LooseCoil" )
      Coil( "S_LooseCoil_bit" )
   END_RUNG
   RUNG wire#powerrail
      Contact( "S_knife" )
      Coil( "S_knife_bit" )
   END_RUNG
   // the same network as SCL:
   "S_Horizontalsealer_bit" := "S_Horizontalsealer";
   "S_Photocell_bit" := "S_Photocell";
   "S_Reedlvl_bit" := "S_Reedlvl";
   "S_OpenDoor_bit" := "S_OpenDoor";
   "S_StuckCoil_bit" := "S_StuckCoil";
   "S_UnwinderOn_bit" := "S_UnwinderOn";
   "S_UnwinderOff_bit" := "S_UnwinderOff";
   "S_LooseCoil_bit" := "S_LooseCoil";
   "S_knife_bit" := "S_knife";
END_REGION

REGION Network 6: Peripherals EV
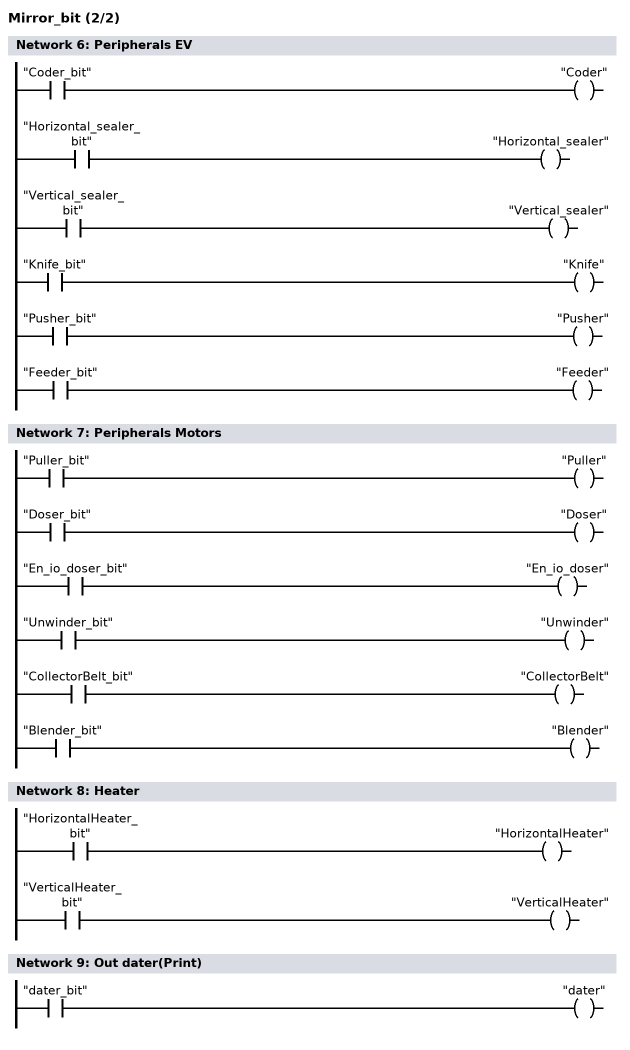
   RUNG wire#powerrail
      Contact( "Coder_bit" )
      Coil( "Coder" )
   END_RUNG
   RUNG wire#powerrail
      Contact( "Horizontal_sealer_bit" )
      Coil( "Horizontal_sealer" )
   END_RUNG
   RUNG wire#powerrail
      Contact( "Vertical_sealer_bit" )
      Coil( "Vertical_sealer" )
   END_RUNG
   RUNG wire#powerrail
      Contact( "Knife_bit" )
      Coil( "Knife" )
   END_RUNG
   RUNG wire#powerrail
      Contact( "Pusher_bit" )
      Coil( "Pusher" )
   END_RUNG
   RUNG wire#powerrail
      Contact( "Feeder_bit" )
      Coil( "Feeder" )
   END_RUNG
   // the same network as SCL:
   "Coder" := "Coder_bit";
   "Horizontal_sealer" := "Horizontal_sealer_bit";
   "Vertical_sealer" := "Vertical_sealer_bit";
   "Knife" := "Knife_bit";
   "Pusher" := "Pusher_bit";
   "Feeder" := "Feeder_bit";
END_REGION

REGION Network 7: Peripherals Motors
   RUNG wire#powerrail
      Contact( "Puller_bit" )
      Coil( "Puller" )
   END_RUNG
   RUNG wire#powerrail
      Contact( "Doser_bit" )
      Coil( "Doser" )
   END_RUNG
   RUNG wire#powerrail
      Contact( "En_io_doser_bit" )
      Coil( "En_io_doser" )
   END_RUNG
   RUNG wire#powerrail
      Contact( "Unwinder_bit" )
      Coil( "Unwinder" )
   END_RUNG
   RUNG wire#powerrail
      Contact( "CollectorBelt_bit" )
      Coil( "CollectorBelt" )
   END_RUNG
   RUNG wire#powerrail
      Contact( "Blender_bit" )
      Coil( "Blender" )
   END_RUNG
   // the same network as SCL:
   "Puller" := "Puller_bit";
   "Doser" := "Doser_bit";
   "En_io_doser" := "En_io_doser_bit";
   "Unwinder" := "Unwinder_bit";
   "CollectorBelt" := "CollectorBelt_bit";
   "Blender" := "Blender_bit";
END_REGION

REGION Network 8: Heater
   RUNG wire#powerrail
      Contact( "HorizontalHeater_bit" )
      Coil( "HorizontalHeater" )
   END_RUNG
   RUNG wire#powerrail
      Contact( "VerticalHeater_bit" )
      Coil( "VerticalHeater" )
   END_RUNG
   // the same network as SCL:
   "HorizontalHeater" := "HorizontalHeater_bit";
   "VerticalHeater" := "VerticalHeater_bit";
END_REGION

REGION Network 9: Out dater(Print)
   RUNG wire#powerrail
      Contact( "dater_bit" )
      Coil( "dater" )
   END_RUNG
   // the same network as SCL:
   "dater" := "dater_bit";
END_REGION
END_ORGANIZATION_BLOCK

ORGANIZATION_BLOCK "Stages"   // OB127, LAD, ProgramCycle
TITLE = "Main Program Sweep (Cycle)"
{ S7_Optimized_Access := 'TRUE' }
VERSION : 0.1
   VAR_INPUT
      Initial_Call : Bool;   // Initial call of this OB
      Remanence : Bool;   // =True, if remanent data are available
   END_VAR
   VAR_TEMP   // added for the SCL form of the ladder/FBD networks
      _w1 : Bool;
      _w2 : Bool;
   END_VAR
BEGIN

REGION Network 1: Etapa de Paro de maquina
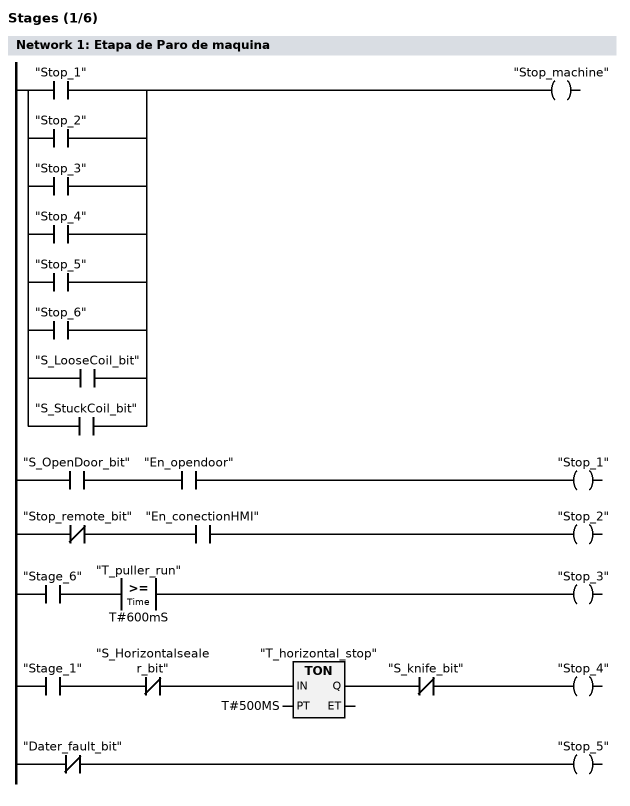
   "Stop_machine" := "Stop_1" OR "Stop_2" OR "Stop_3" OR "Stop_4" OR "Stop_5" OR "Stop_6" OR "S_LooseCoil_bit" OR "S_StuckCoil_bit";
   "Stop_1" := "S_OpenDoor_bit" AND "En_opendoor";
   "Stop_2" := NOT "Stop_remote_bit" AND "En_conectionHMI";
   "Stop_3" := "Stage_6" AND ("T_puller_run" >= T#600mS);
   "T_horizontal_stop".TON(IN := "Stage_1" AND NOT "S_Horizontalsealer_bit", PT := T#500MS);
   "Stop_4" := "T_horizontal_stop".Q AND NOT "S_knife_bit";
   "Stop_5" := NOT "Dater_fault_bit";
END_REGION

REGION Network 2: Etapa de Reinicio
   // mover etapas individuales Como stage blender
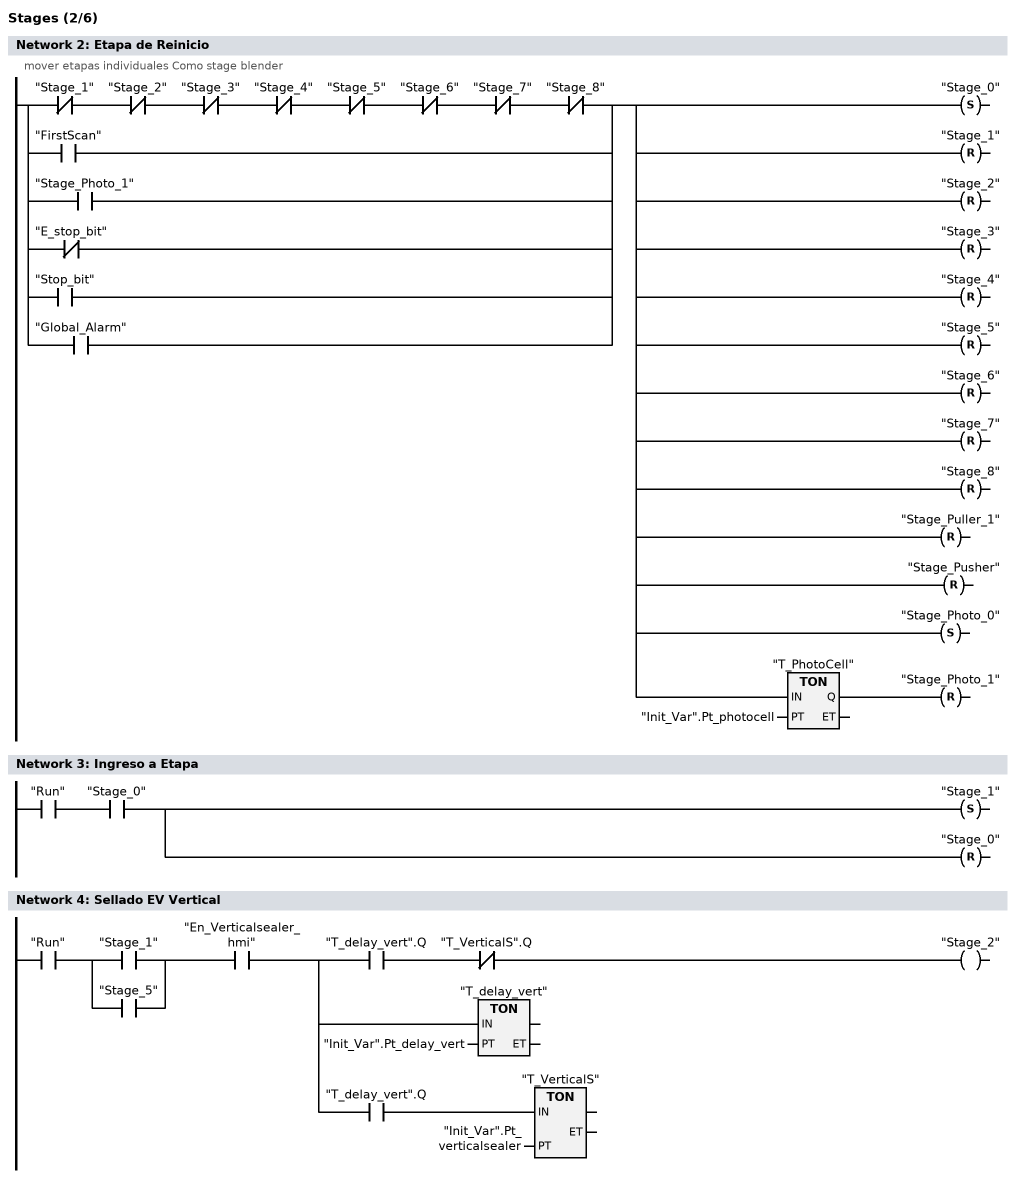
   #_w1 := (NOT "Stage_1" AND NOT "Stage_2" AND NOT "Stage_3" AND NOT "Stage_4" AND NOT "Stage_5" AND NOT "Stage_6" AND NOT "Stage_7" AND NOT "Stage_8") OR "FirstScan" OR "Stage_Photo_1" OR NOT "E_stop_bit" OR "Stop_bit" OR "Global_Alarm";
   IF #_w1 THEN
       "Stage_0" := TRUE;
       "Stage_1" := FALSE;
       "Stage_2" := FALSE;
       "Stage_3" := FALSE;
       "Stage_4" := FALSE;
       "Stage_5" := FALSE;
       "Stage_6" := FALSE;
       "Stage_7" := FALSE;
       "Stage_8" := FALSE;
       "Stage_Puller_1" := FALSE;
       "Stage_Pusher" := FALSE;
       "Stage_Photo_0" := TRUE;
   END_IF;
   "T_PhotoCell".TON(IN := #_w1, PT := "Init_Var".Pt_photocell);
   IF "T_PhotoCell".Q THEN "Stage_Photo_1" := FALSE; END_IF;
END_REGION

REGION Network 3: Ingreso a Etapa
   RUNG wire#powerrail
      Contact( "Run" )
      Contact( "Stage_0" )
      wire#w1
      S_Coil( "Stage_1" )
   END_RUNG
   RUNG wire#w1
      R_Coil( "Stage_0" )
   END_RUNG
   // the same network as SCL:
   IF "Run" AND "Stage_0" THEN
       "Stage_1" := TRUE;
       "Stage_0" := FALSE;
   END_IF;
END_REGION

REGION Network 4: Sellado EV Vertical
   #_w1 := "Run" AND ("Stage_1" OR "Stage_5") AND "En_Verticalsealer_hmi";
   "Stage_2" := #_w1 AND "T_delay_vert".Q AND NOT "T_VerticalS".Q;
   "T_delay_vert".TON(IN := #_w1, PT := "Init_Var".Pt_delay_vert);
   "T_VerticalS".TON(IN := #_w1 AND "T_delay_vert".Q, PT := "Init_Var".Pt_verticalsealer);
END_REGION

REGION Network 5: Sellado EV Horizontal
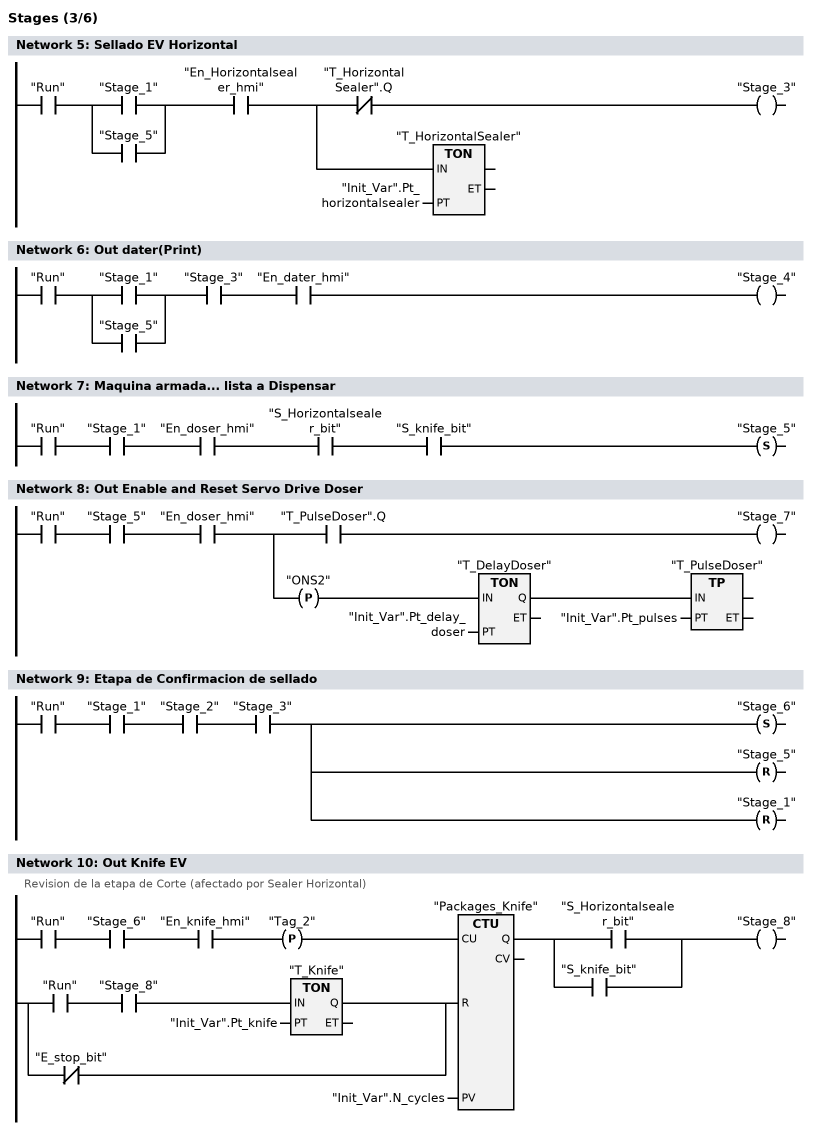
   #_w1 := "Run" AND ("Stage_1" OR "Stage_5") AND "En_Horizontalsealer_hmi";
   "Stage_3" := #_w1 AND NOT "T_HorizontalSealer".Q;
   "T_HorizontalSealer".TON(IN := #_w1, PT := "Init_Var".Pt_horizontalsealer);
END_REGION

REGION Network 6: Out dater(Print)
   RUNG wire#powerrail
      Contact( "Run" )
      wire#w1
      Contact( "Stage_1" )
      wire#w2
      Contact( "Stage_3" )
      Contact( "En_dater_hmi" )
      Coil( "Stage_4" )
   END_RUNG
   RUNG wire#w1
      Contact( "Stage_5" )
   END_RUNG wire#w2
   // the same network as SCL:
   "Stage_4" := "Run" AND ("Stage_1" OR "Stage_5") AND "Stage_3" AND "En_dater_hmi";
END_REGION

REGION Network 7: Maquina armada... lista a Dispensar
   RUNG wire#powerrail
      Contact( "Run" )
      Contact( "Stage_1" )
      Contact( "En_doser_hmi" )
      Contact( "S_Horizontalsealer_bit" )
      Contact( "S_knife_bit" )
      S_Coil( "Stage_5" )
   END_RUNG
   // the same network as SCL:
   IF "Run" AND "Stage_1" AND "En_doser_hmi" AND "S_Horizontalsealer_bit" AND "S_knife_bit" THEN
       "Stage_5" := TRUE;
   END_IF;
END_REGION

REGION Network 8: Out Enable and Reset Servo Drive Doser
   #_w1 := "Run" AND "Stage_5" AND "En_doser_hmi";
   "Stage_7" := #_w1 AND "T_PulseDoser".Q;
   #_w2 := #_w1 AND NOT "ONS2";   // rising edge
   "ONS2" := #_w1;
   "T_DelayDoser".TON(IN := #_w2, PT := "Init_Var".Pt_delay_doser);
   "T_PulseDoser".TP(IN := "T_DelayDoser".Q, PT := "Init_Var".Pt_pulses);
END_REGION

REGION Network 9: Etapa de Confirmacion de sellado
   RUNG wire#powerrail
      Contact( "Run" )
      Contact( "Stage_1" )
      Contact( "Stage_2" )
      Contact( "Stage_3" )
      wire#w1
      S_Coil( "Stage_6" )
   END_RUNG
   RUNG wire#w1
      R_Coil( "Stage_5" )
   END_RUNG
   RUNG wire#w1
      R_Coil( "Stage_1" )
   END_RUNG
   // the same network as SCL:
   IF "Run" AND "Stage_1" AND "Stage_2" AND "Stage_3" THEN
       "Stage_6" := TRUE;
       "Stage_5" := FALSE;
       "Stage_1" := FALSE;
   END_IF;
END_REGION

REGION Network 10: Out Knife EV
   // Revision de la etapa de Corte (afectado por Sealer Horizontal)
   #_w1 := "Run" AND "Stage_6" AND "En_knife_hmi";
   #_w2 := #_w1 AND NOT "Tag_2";   // rising edge
   "Tag_2" := #_w1;
   "T_Knife".TON(IN := "Run" AND "Stage_8", PT := "Init_Var".Pt_knife);
   "Packages_Knife".CTU(CU := #_w2, R := "T_Knife".Q OR NOT "E_stop_bit", PV := "Init_Var".N_cycles);
   "Stage_8" := "Packages_Knife".Q AND ("S_Horizontalsealer_bit" OR "S_knife_bit");
END_REGION

REGION Network 11
   // Revision de la etapa de Corte (afecta puller)
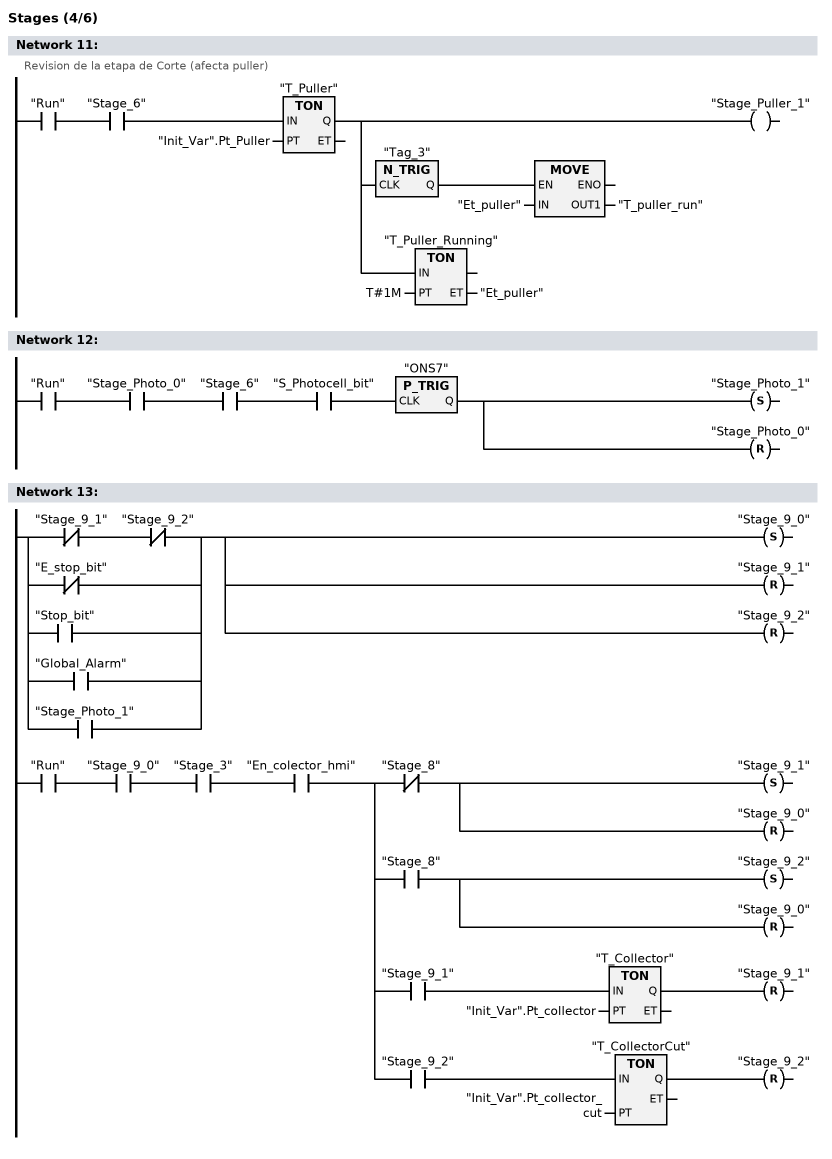
   "T_Puller".TON(IN := "Run" AND "Stage_6", PT := "Init_Var".Pt_Puller);
   "Stage_Puller_1" := "T_Puller".Q;
   #_w1 := NOT "T_Puller".Q AND "Tag_3";   // falling edge
   "Tag_3" := "T_Puller".Q;
   IF #_w1 THEN "T_puller_run" := "Et_puller"; END_IF;
   "T_Puller_Running".TON(IN := "T_Puller".Q, PT := T#1M, ET => "Et_puller");
END_REGION

REGION Network 12
   RUNG wire#powerrail
      Contact( "Run" )
      Contact( "Stage_Photo_0" )
      Contact( "Stage_6" )
      Contact( "S_Photocell_bit" )
      P_Trig( "ONS7" )
      wire#w1
      S_Coil( "Stage_Photo_1" )
   END_RUNG
   RUNG wire#w1
      R_Coil( "Stage_Photo_0" )
   END_RUNG
   // the same network as SCL:
   #_w1 := "Run" AND "Stage_Photo_0" AND "Stage_6" AND "S_Photocell_bit";
   #_w2 := #_w1 AND NOT "ONS7";   // rising edge
   "ONS7" := #_w1;
   IF #_w2 THEN
       "Stage_Photo_1" := TRUE;
       "Stage_Photo_0" := FALSE;
   END_IF;
END_REGION

REGION Network 13
   IF (NOT "Stage_9_1" AND NOT "Stage_9_2") OR NOT "E_stop_bit" OR "Stop_bit" OR "Global_Alarm" OR "Stage_Photo_1" THEN
       "Stage_9_0" := TRUE;
   END_IF;
   #_w1 := (NOT "Stage_9_1" AND NOT "Stage_9_2") OR NOT "E_stop_bit" OR "Stop_bit" OR "Global_Alarm" OR "Stage_Photo_1";
   IF #_w1 THEN
       "Stage_9_1" := FALSE;
       "Stage_9_2" := FALSE;
   END_IF;
   #_w2 := "Run" AND "Stage_9_0" AND "Stage_3" AND "En_colector_hmi";
   IF #_w2 AND NOT "Stage_8" THEN
       "Stage_9_1" := TRUE;
       "Stage_9_0" := FALSE;
   END_IF;
   IF #_w2 AND "Stage_8" THEN
       "Stage_9_2" := TRUE;
       "Stage_9_0" := FALSE;
   END_IF;
   "T_Collector".TON(IN := #_w2 AND "Stage_9_1", PT := "Init_Var".Pt_collector);
   IF "T_Collector".Q THEN "Stage_9_1" := FALSE; END_IF;
   "T_CollectorCut".TON(IN := #_w2 AND "Stage_9_2", PT := "Init_Var".Pt_collector_cut);
   IF "T_CollectorCut".Q THEN "Stage_9_2" := FALSE; END_IF;
END_REGION

REGION Network 14
   // feed
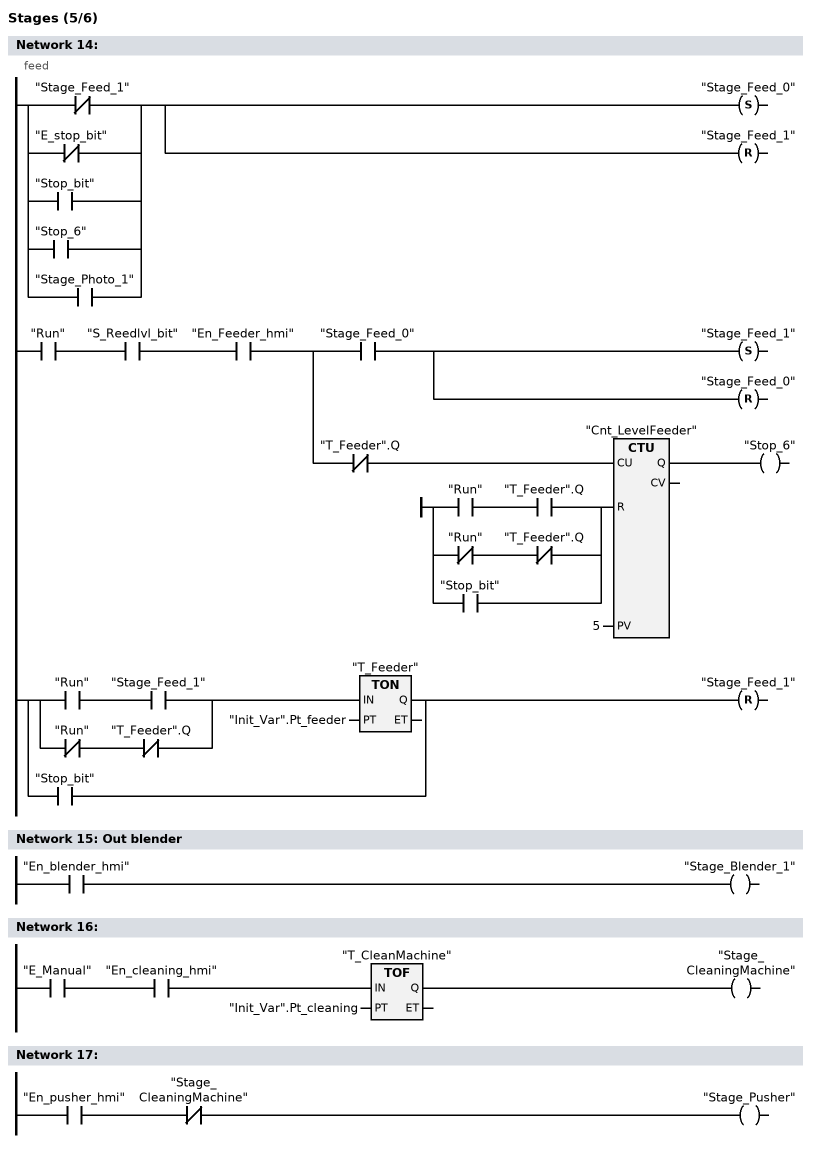
   IF NOT "Stage_Feed_1" OR NOT "E_stop_bit" OR "Stop_bit" OR "Stop_6" OR "Stage_Photo_1" THEN
       "Stage_Feed_0" := TRUE;
       "Stage_Feed_1" := FALSE;
   END_IF;
   #_w1 := "Run" AND "S_Reedlvl_bit" AND "En_Feeder_hmi";
   IF #_w1 AND "Stage_Feed_0" THEN
       "Stage_Feed_1" := TRUE;
       "Stage_Feed_0" := FALSE;
   END_IF;
   "Cnt_LevelFeeder".CTU(CU := #_w1 AND NOT "T_Feeder".Q,
                         R := ("Run" AND "T_Feeder".Q) OR (NOT "Run" AND NOT "T_Feeder".Q) OR "Stop_bit",
                         PV := 5);
   "Stop_6" := "Cnt_LevelFeeder".Q;
   "T_Feeder".TON(IN := ("Run" AND "Stage_Feed_1") OR (NOT "Run" AND NOT "T_Feeder".Q),
                  PT := "Init_Var".Pt_feeder);
   IF "T_Feeder".Q OR "Stop_bit" THEN "Stage_Feed_1" := FALSE; END_IF;
END_REGION

REGION Network 15: Out blender
   RUNG wire#powerrail
      Contact( "En_blender_hmi" )
      Coil( "Stage_Blender_1" )
   END_RUNG
   // the same network as SCL:
   "Stage_Blender_1" := "En_blender_hmi";
END_REGION

REGION Network 16
   "T_CleanMachine".TOF(IN := "E_Manual" AND "En_cleaning_hmi", PT := "Init_Var".Pt_cleaning);
   "Stage_CleaningMachine" := "T_CleanMachine".Q;
END_REGION

REGION Network 17
   RUNG wire#powerrail
      Contact( "En_pusher_hmi" )
      I_Contact( "Stage_CleaningMachine" )
      Coil( "Stage_Pusher" )
   END_RUNG
   // the same network as SCL:
   "Stage_Pusher" := "En_pusher_hmi" AND NOT "Stage_CleaningMachine";
END_REGION

REGION Network 18
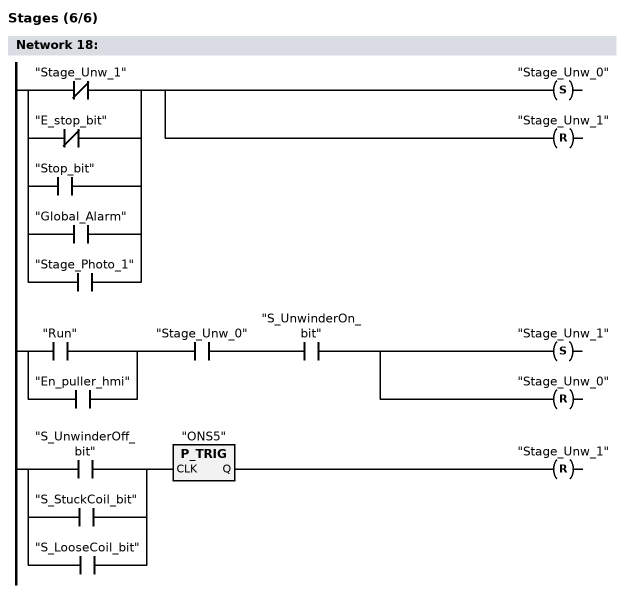
   RUNG wire#powerrail
      I_Contact( "Stage_Unw_1" )
      wire#w1
      S_Coil( "Stage_Unw_0" )
   END_RUNG
   RUNG wire#powerrail
      I_Contact( "E_stop_bit" )
   END_RUNG wire#w1
   RUNG wire#powerrail
      Contact( "Stop_bit" )
   END_RUNG wire#w1
   RUNG wire#powerrail
      Contact( "Global_Alarm" )
   END_RUNG wire#w1
   RUNG wire#powerrail
      Contact( "Stage_Photo_1" )
   END_RUNG wire#w1
   RUNG wire#w1
      R_Coil( "Stage_Unw_1" )
   END_RUNG
   RUNG wire#powerrail
      Contact( "Run" )
      wire#w2
      Contact( "Stage_Unw_0" )
      Contact( "S_UnwinderOn_bit" )
      wire#w3
      S_Coil( "Stage_Unw_1" )
   END_RUNG
   RUNG wire#powerrail
      Contact( "En_puller_hmi" )
   END_RUNG wire#w2
   RUNG wire#w3
      R_Coil( "Stage_Unw_0" )
   END_RUNG
   RUNG wire#powerrail
      Contact( "S_UnwinderOff_bit" )
      wire#w4
      P_Trig( "ONS5" )
      R_Coil( "Stage_Unw_1" )
   END_RUNG
   RUNG wire#powerrail
      Contact( "S_StuckCoil_bit" )
   END_RUNG wire#w4
   RUNG wire#powerrail
      Contact( "S_LooseCoil_bit" )
   END_RUNG wire#w4
   // the same network as SCL:
   IF NOT "Stage_Unw_1" OR NOT "E_stop_bit" OR "Stop_bit" OR "Global_Alarm" OR "Stage_Photo_1" THEN
       "Stage_Unw_0" := TRUE;
       "Stage_Unw_1" := FALSE;
   END_IF;
   IF ("Run" OR "En_puller_hmi") AND "Stage_Unw_0" AND "S_UnwinderOn_bit" THEN
       "Stage_Unw_1" := TRUE;
       "Stage_Unw_0" := FALSE;
   END_IF;
   #_w1 := "S_UnwinderOff_bit" OR "S_StuckCoil_bit" OR "S_LooseCoil_bit";
   #_w2 := #_w1 AND NOT "ONS5";   // rising edge
   "ONS5" := #_w1;
   IF #_w2 THEN "Stage_Unw_1" := FALSE; END_IF;
END_REGION
END_ORGANIZATION_BLOCK

(* ===== HMI "HMI_RT_1" =====
system functions are stored by id; their names below are inferred from use
connection "HMI_Connection_1": ETHERNET, SMART_S7_1200_OMS

HMI tags "Default tag table"
   "Tag_ScreenNumber" : UInt, internal
   "HMI_Alarms" : UInt AT %DB1.DBW0, 1 s
   "En_opendoor" : Bool = PLC En_opendoor AT %M15.0, 1 s
   "En_conectionHMI" : Bool = PLC En_conectionHMI AT %M15.7, 1 s
   "Init_Var_Pt_coder" : Time = PLC Init_Var.Pt_coder, 1 s
   "Init_Var_Pt_horizontalsealer" : Time = PLC Init_Var.Pt_horizontalsealer, 1 s
   "Init_Var_Pt_verticalsealer" : Time = PLC Init_Var.Pt_verticalsealer, 1 s
   "Init_Var_Pt_delay_vert" : Time = PLC Init_Var.Pt_delay_vert, 1 s
   "Init_Var_Pt_collector" : Time = PLC Init_Var.Pt_collector, 1 s
   "Init_Var_Pt_collector_cut" : Time = PLC Init_Var.Pt_collector_cut, 1 s
   "Init_Var_Pt_pulses" : Time = PLC Init_Var.Pt_pulses, 1 s
   "Init_Var_Pt_delay_doser" : Time = PLC Init_Var.Pt_delay_doser, 1 s
   "Init_Var_Pt_photocell" : Time = PLC Init_Var.Pt_photocell, 1 s
   "Init_Var_Pt_knife" : Time = PLC Init_Var.Pt_knife, 1 s
   "Init_Var_Pt_Puller" : Time = PLC Init_Var.Pt_Puller, 1 s
   "Init_Var_Pt_feeder" : Time = PLC Init_Var.Pt_feeder, 1 s
   "Init_Var_N_cycles" : Int = PLC Init_Var.N_cycles, 1 s
   "En_Verticalsealer_hmi" : Bool = PLC En_Verticalsealer_hmi AT %M21.1, 1 s
   "TestVerticalsealer_hmi" : Bool = PLC TestVerticalsealer_hmi AT %M21.2, 1 s
   "En_Horizontalsealer_hmi" : Bool = PLC En_Horizontalsealer_hmi AT %M21.3, 1 s
   "En_doser_hmi" : Bool = PLC En_doser_hmi AT %M21.7, 1 s
   "En_dater_hmi" : Bool = PLC En_dater_hmi AT %M21.5, 1 s
   "En_knife_hmi" : Bool = PLC En_knife_hmi AT %M22.0, 1 s
   "Testhorizontalsealer_hmi" : Bool = PLC Testhorizontalsealer_hmi AT %M21.4, 1 s
   "Testdater_hmi" : Bool = PLC Testdater_hmi AT %M21.6, 1 s
   "TestKnife_hmi" : Bool = PLC TestKnife_hmi AT %M22.2, 1 s
   "TestCollector_hmi" : Bool = PLC TestCollector_hmi AT %M23.2, 1 s
   "Testdoser_hmi" : Bool = PLC Testdoser_hmi AT %M22.7, 1 s
   "En_Feeder_hmi" : Bool = PLC En_Feeder_hmi AT %M23.3, 1 s
   "En_blender_hmi" : Bool = PLC En_blender_hmi AT %M23.7, 1 s
   "En_cleaning_hmi" : Bool = PLC En_cleaning_hmi AT %M24.2, 1 s
   "Init_Var_Pt_cleaning" : Time = PLC Init_Var.Pt_cleaning, 1 s
   "En_pusher_hmi" : Bool = PLC En_pusher_hmi AT %M24.1, 1 s
   "En_horizontalheater_hmi" : Bool = PLC En_horizontalheater_hmi AT %M24.6, 1 s
   "En_verticalheater_hmi" : Bool = PLC En_verticalheater_hmi AT %M24.7, 1 s
   "TestBlender_hmi" : Bool = PLC TestBlender_hmi AT %M24.0, 1 s
   "PPM" : Int = PLC PPM AT %MW36, 1 s
   "stimate_ppm" : DInt = PLC stimate_ppm AT %MD46, 1 s
   "write_time" : Bool = PLC write_time AT %M56.1, 1 s
   "En_colector_hmi" : Bool = PLC En_colector_hmi AT %M23.1, 1 s
   "En_puller_hmi" : Bool = PLC En_puller_hmi AT %M25.4, 1 s
   "TestPuller_hmi" : Bool = PLC TestPuller_hmi AT %M31.1, 1 s
   "TestFeeder_hmi" : Bool = PLC TestFeeder_hmi AT %M23.6, 1 s
   "db_time_sync_time_local_READ" : DTL = PLC db_time_sync.time_local_READ, 1 s
   "db_time_sync_time_system_READ" : DTL = PLC db_time_sync.time_system_READ, 1 s
   "db_time_sync_time_system_WRITE" : DTL = PLC db_time_sync.time_system_WRITE, 1 s

discrete alarms
   1: 'Alarma activa', class Errors, trigger "HMI_Alarms" bit 8
   2: 'Paro de emergencia activo', class Errors, trigger "HMI_Alarms" bit 9
   3: 'Disparo térmico del motor colector', class Errors, trigger "HMI_Alarms" bit 10
   4: 'Disparo térmico del motor arrastre', class Errors, trigger "HMI_Alarms" bit 11
   5: 'Disparo térmico del motor de bobina', class Errors, trigger "HMI_Alarms" bit 12
   6: 'Servomotor en falla', class Errors, trigger "HMI_Alarms" bit 13
   7: 'Disparo térmico del motor agitador', class Errors, trigger "HMI_Alarms" bit 14
   8: 'Puertas abiertas', class Errors, trigger "HMI_Alarms" bit 15
   9: 'Paro remoto', class Errors, trigger "HMI_Alarms" bit 0
   10: 'Tolva sin producto', class Errors, trigger "HMI_Alarms" bit 1
   11: 'Sello horizontal bloqueado', class Errors, trigger "HMI_Alarms" bit 2
   12: 'Bobina floja', class Errors, trigger "HMI_Alarms" bit 3
   13: 'Bobina atascada', class Errors, trigger "HMI_Alarms" bit 4
   14: 'Falla en fotocelda', class Errors, trigger "HMI_Alarms" bit 5
   15: 'Falla en el codificador', class Errors, trigger "HMI_Alarms" bit 6
   16: 'Falta de producto en tolva', class Errors, trigger "HMI_Alarms" bit 7

Template "Template_1" 800x480
   Button "Exit" at 714,429 size 71x50; TextOff 'Exit'; PictureOff "ExitRuntime_KTP700_Basic_PN_TR"; PictureOn "ExitRuntime_KTP700_Basic_PN_TR"
      on Release: StopRuntime(0)
   Button "Template_Button" at 614,429 size 71x50; TextOff 'Text'; PictureOff "Graphic_2"
      on Release: ActivateScreen("Support", 0)
   Button "Template_Button_1" at 514,429 size 71x50; TextOff 'Text'
   Button "Template_Button_2" at 414,429 size 71x50; TextOff 'Text'
   Button "Template_Button_3" at 314,429 size 71x50; TextOff 'Text'; PictureOff "Graphic_4"
      on Release: ActivateScreen("Test", 0)
   Button "Template_Button_4" at 214,429 size 71x50; TextOff 'Text'; PictureOff "Graphic_3"
      on Release: ActivateScreen("Production", 0)
   Button "Alarms" at 114,429 size 71x50; TextOff 'Alarms'; PictureOff "AlarmDisplay_KTP700_Basic_PN_TR"; PictureOn "AlarmDisplay_KTP700_Basic_PN_TR"
      on Release: ActivateScreen("Alarms", 0)
   Button "Start screen" at 14,429 size 71x50; TextOff 'Start screen'; PictureOff "NavigateHome_KTP700_Basic_PN_TR"; PictureOn "NavigateHome_KTP700_Basic_PN_TR"
      on Release: ActivateScreen("Home", 0)
   SymbolicIOField "Symbolic_IO_Field_Screen" at 93,9 size 600x33; TextOff '0'; TextOn '1'; TextList "TextList_ScreenNames"
      ProcessValue <- "Tag_ScreenNumber"
      on Change: ActivateScreenByNumber("Tag_ScreenNumber", 0)
   DateTimeField "HmiScreenItemData" at 695,25 size 105x25
   DateTimeField "HmiScreenItemData_1" at 695,0 size 105x25
   GraphicView "Logo" at 0,0 size 90x65; Picture "Cafesoluble-300x300 copy"
   Softkey "Softkey_F1" at 0,0 size 0x0
      on KeyUp: ActivateScreen("Home", 0)
   Softkey "Softkey_F2" at 0,0 size 0x0
      on KeyUp: ActivateScreen("Alarms", 0)
   Softkey "Softkey_F3" at 0,0 size 0x0
      on KeyUp: ActivateScreen("Production", 0)
   Softkey "Softkey_F4" at 0,0 size 0x0
      on KeyUp: ActivateScreen("Test", 0)
   Softkey "Softkey_F7" at 0,0 size 0x0
      on KeyUp: ActivateScreen("Support", 0)

screen "Home" 800x480, template "Template_1"
   on GenerateScreen: SetTag("Tag_ScreenNumber", 1)
   TextField "HmiScreenItemData" at 18,348 size 171x28; Text 'Llenadora'
   GraphicView "Graphic view_1" at 0,85 size 366x261; Picture "LOGO-CSSA-1"
   TextField "HmiScreenItemData_2" at 18,372 size 171x28; Text 'Código'
   TextField "HmiScreenItemData_1" at 226,348 size 524x28; Text 'SpeedBag 4000'
   TextField "HmiScreenItemData_3" at 226,372 size 524x28; Text 'EB23'
   Button "HmiScreenItemData_9" at 529,82 size 130x50; TextOn 'SIMATIC PLC system diagnostics'; TextOff 'Limpieza'; PictureOn "Navigates to SIMATIC PLC system diagnostics for HMI_1"; PictureOff "Navigates to SIMATIC PLC system diagnostics for HMI_1"
      on Press: function_b14e0dd5("En_cleaning_hmi", 0)
      Appearance <- "En_cleaning_hmi"
   IOField "I/O field_15" at 668,82 size 80x50; FormatPattern 99999
      ProcessValue <- "Init_Var_Pt_cleaning"
   Button "HmiScreenItemData_4" at 529,138 size 130x50; TextOn 'SIMATIC PLC system diagnostics'; TextOff 'P.P.M real'; PictureOn "Navigates to SIMATIC PLC system diagnostics for HMI_1"; PictureOff "Navigates to SIMATIC PLC system diagnostics for HMI_1"
   IOField "I/O field_1" at 668,138 size 80x50; FormatPattern 99999
      ProcessValue <- "PPM"
   Button "HmiScreenItemData_5" at 529,194 size 130x50; TextOn 'SIMATIC PLC system diagnostics'; TextOff 'P.P.M calculado'; PictureOn "Navigates to SIMATIC PLC system diagnostics for HMI_1"; PictureOff "Navigates to SIMATIC PLC system diagnostics for HMI_1"
      ProcessValue <- "stimate_ppm"
   IOField "I/O field_2" at 668,194 size 80x50; FormatPattern 9999999999
      ProcessValue <- "stimate_ppm"

screen "Alarms" 800x480, template "Template_1"
   on GenerateScreen: SetTag("Tag_ScreenNumber", 2)
   AlarmView "Alarm view_1" at 3,70 size 792x349

screen "Production" 800x480, template "Template_1"
   on GenerateScreen: SetTag("Tag_ScreenNumber", 3)
   Button "HmiScreenItemData_1" at 17,156 size 130x50; TextOn 'SIMATIC PLC system diagnostics'; TextOff 'S. horizontal'; PictureOn "Navigates to SIMATIC PLC system diagnostics for HMI_1"; PictureOff "Navigates to SIMATIC PLC system diagnostics for HMI_1"
      on Press: InvertBit("En_Horizontalsealer_hmi")
      Appearance <- "En_Horizontalsealer_hmi"
   IOField "I/O field_1" at 155,156 size 80x50; FormatPattern 99999
      ProcessValue <- "Init_Var_Pt_horizontalsealer"
   Button "HmiScreenItemData_2" at 340,156 size 130x50; TextOn 'SIMATIC PLC system diagnostics'; TextOff 'Cuchilla'; PictureOn "Navigates to SIMATIC PLC system diagnostics for HMI_1"; PictureOff "Navigates to SIMATIC PLC system diagnostics for HMI_1"
      on Press: InvertBit("En_knife_hmi")
      Appearance <- "En_knife_hmi"
   IOField "I/O field_3" at 481,156 size 80x50; FormatPattern 99999
      ProcessValue <- "Init_Var_Pt_knife"
   Button "HmiScreenItemData_3" at 17,212 size 130x50; TextOn 'SIMATIC PLC system diagnostics'; TextOff 'S. vertical'; PictureOn "Navigates to SIMATIC PLC system diagnostics for HMI_1"; PictureOff "Navigates to SIMATIC PLC system diagnostics for HMI_1"
      on Press: InvertBit("En_Verticalsealer_hmi")
      Appearance <- "En_Verticalsealer_hmi"
   IOField "I/O field_5" at 155,212 size 80x50; FormatPattern 99999
      ProcessValue <- "Init_Var_Pt_verticalsealer"
   Button "HmiScreenItemData_4" at 17,100 size 130x50; TextOn 'SIMATIC PLC system diagnostics'; TextOff 'Codificador'; PictureOn "Navigates to SIMATIC PLC system diagnostics for HMI_1"; PictureOff "Navigates to SIMATIC PLC system diagnostics for HMI_1"
      on Press: InvertBit("En_dater_hmi")
      Appearance <- "En_dater_hmi"
   Button "HmiScreenItemData_5" at 340,212 size 130x50; TextOn 'SIMATIC PLC system diagnostics'; TextOff 'Banda arrastre'; PictureOn "Navigates to SIMATIC PLC system diagnostics for HMI_1"; PictureOff "Navigates to SIMATIC PLC system diagnostics for HMI_1"
      on Press: InvertBit("En_puller_hmi")
      Appearance <- "En_puller_hmi"
   Button "HmiScreenItemData_6" at 17,324 size 130x50; TextOn 'SIMATIC PLC system diagnostics'; TextOff 'Dosificador'; PictureOn "Navigates to SIMATIC PLC system diagnostics for HMI_1"; PictureOff "Navigates to SIMATIC PLC system diagnostics for HMI_1"
      on Press: InvertBit("En_doser_hmi")
      Appearance <- "En_doser_hmi"
   IOField "I/O field_12" at 155,324 size 80x50; FormatPattern 99999
      ProcessValue <- "Init_Var_Pt_pulses"
   TextField "Text field_1" at 151,61 size 88x23; Text 'Encendido'
   Button "HmiScreenItemData_7" at 340,100 size 130x50; TextOn 'SIMATIC PLC system diagnostics'; TextOff 'Fotocelda'; PictureOn "Navigates to SIMATIC PLC system diagnostics for HMI_1"; PictureOff "Navigates to SIMATIC PLC system diagnostics for HMI_1"
   IOField "I/O field_13" at 481,100 size 80x50; FormatPattern 99999
      ProcessValue <- "Init_Var_Pt_photocell"
   TextField "Text field_3" at 46,61 size 92x23; Text 'Parámetro'
   Button "HmiScreenItemData_10" at 630,252 size 130x50; TextOn 'SIMATIC PLC system diagnostics'; TextOff 'Presionador'; PictureOn "Navigates to SIMATIC PLC system diagnostics for HMI_1"; PictureOff "Navigates to SIMATIC PLC system diagnostics for HMI_1"
      on Press: InvertBit("En_pusher_hmi")
      Appearance <- "En_pusher_hmi"
   IOField "I/O field_2" at 155,100 size 80x50; FormatPattern 99999
      ProcessValue <- "Init_Var_Pt_coder"
   Button "HmiScreenItemData_8" at 631,84 size 130x50; TextOn 'SIMATIC PLC system diagnostics'; TextOff 'T. Horizontal'; PictureOn "Navigates to SIMATIC PLC system diagnostics for HMI_1"; PictureOff "Navigates to SIMATIC PLC system diagnostics for HMI_1"
      on Press: InvertBit("En_horizontalheater_hmi")
      Appearance <- "En_horizontalheater_hmi"
   Button "HmiScreenItemData_11" at 631,140 size 130x50; TextOn 'SIMATIC PLC system diagnostics'; TextOff 'T. Vertical'; PictureOn "Navigates to SIMATIC PLC system diagnostics for HMI_1"; PictureOff "Navigates to SIMATIC PLC system diagnostics for HMI_1"
      on Press: InvertBit("En_verticalheater_hmi")
      Appearance <- "En_verticalheater_hmi"
   Button "HmiScreenItemData_12" at 340,268 size 130x50; TextOn 'SIMATIC PLC system diagnostics'; TextOff 'Producto'; PictureOn "Navigates to SIMATIC PLC system diagnostics for HMI_1"; PictureOff "Navigates to SIMATIC PLC system diagnostics for HMI_1"
      on Press: InvertBit("En_Feeder_hmi")
      Appearance <- "En_Feeder_hmi"
   Button "HmiScreenItemData_13" at 630,196 size 130x50; TextOn 'SIMATIC PLC system diagnostics'; TextOff 'Agitador'; PictureOn "Navigates to SIMATIC PLC system diagnostics for HMI_1"; PictureOff "Navigates to SIMATIC PLC system diagnostics for HMI_1"
      on Press: InvertBit("En_blender_hmi")
      Appearance <- "En_blender_hmi"
   Button "HmiScreenItemData_15" at 17,268 size 130x50; TextOn 'SIMATIC PLC system diagnostics'; TextOff 'Colector'; PictureOn "Navigates to SIMATIC PLC system diagnostics for HMI_1"; PictureOff "Navigates to SIMATIC PLC system diagnostics for HMI_1"
      on Press: InvertBit("En_colector_hmi")
      Appearance <- "En_colector_hmi"
   IOField "I/O field_6" at 155,268 size 80x50; FormatPattern 99999
      ProcessValue <- "Init_Var_Pt_collector"
   IOField "I/O field_7" at 244,268 size 80x50; FormatPattern 99999
      ProcessValue <- "Init_Var_Pt_collector_cut"
   IOField "I/O field_8" at 481,268 size 80x50; FormatPattern 999999
      ProcessValue <- "Init_Var_Pt_feeder"
   Button "HmiScreenItemData_16" at 630,308 size 130x50; TextOn 'SIMATIC PLC system diagnostics'; TextOff 'Conexión'; PictureOn "Navigates to SIMATIC PLC system diagnostics for HMI_1"; PictureOff "Navigates to SIMATIC PLC system diagnostics for HMI_1"
      on Press: InvertBit("En_conectionHMI")
      Appearance <- "En_conectionHMI"
   IOField "I/O field_9" at 481,212 size 80x50; FormatPattern 99999
      ProcessValue <- "Init_Var_Pt_Puller"
   IOField "I/O field_10" at 243,212 size 80x50; FormatPattern 99999
      ProcessValue <- "Init_Var_Pt_delay_vert"
   IOField "I/O field_11" at 244,324 size 80x50; FormatPattern 99999
      ProcessValue <- "Init_Var_Pt_delay_doser"
   TextField "Text field_2" at 248,61 size 71x23; Text 'Retardo'
   TextField "Text field_4" at 155,77 size 81x23; Text 'segundos'
   TextField "Text field_6" at 243,77 size 81x23; Text 'segundos'
   Button "HmiScreenItemData_14" at 630,364 size 130x50; TextOn 'SIMATIC PLC system diagnostics'; TextOff 'Puertas'; PictureOn "Navigates to SIMATIC PLC system diagnostics for HMI_1"; PictureOff "Navigates to SIMATIC PLC system diagnostics for HMI_1"
      on Press: InvertBit("En_opendoor")
      Appearance <- "En_opendoor"
   TextField "Text field_5" at 479,61 size 88x23; Text 'Encendido'
   TextField "Text field_7" at 483,77 size 81x23; Text 'segundos'
   TextField "Text field_8" at 366,61 size 92x23; Text 'Parámetro'
   Button "HmiScreenItemData_9" at 340,324 size 130x50; TextOn 'SIMATIC PLC system diagnostics'; TextOff 'Ristra'; PictureOn "Navigates to SIMATIC PLC system diagnostics for HMI_1"; PictureOff "Navigates to SIMATIC PLC system diagnostics for HMI_1"
   IOField "I/O field_4" at 481,324 size 80x50; FormatPattern 99999
      ProcessValue <- "Init_Var_N_cycles"

screen "Support" 800x480, template "Template_1"
   on GenerateScreen: SetTag("Tag_ScreenNumber", 4)
   Button "HmiScreenItemData" at 18,139 size 159x47; TextOn 'Online'; TextOff 'Online'
      on Release: function_bb44b551(0)
   Button "HmiScreenItemData_1" at 18,186 size 159x47; TextOn 'Offline'; TextOff 'Offline'
      on Release: function_bb44b551(1)
   Button "HmiScreenItemData_2" at 18,233 size 159x47; TextOn 'Transfer'; TextOff 'Transfer'
      on Release: function_bb44b551(2)
   Button "HmiScreenItemData_3" at 18,280 size 159x47; TextOn 'Toggle language'; TextOff 'Toggle language'
      on Release: function_fb9197e8(-1)
   GraphicView "Graphic view_1" at 212,72 size 376x249; Picture "Servicios de Consultoría e Ingeniería - Final.fw"
   TextField "Text field_3" at 284,316 size 232x23; Text 'Contacto: info@scisa.com.ni'
   Button "HmiScreenItemData_4" at 18,92 size 159x47; TextOn 'SIMATIC PLC system diagnostics'; TextOff 'SIMATIC PLC system diagnostics'; PictureOn "Navigates to SIMATIC PLC system diagnostics for HMI_1"; PictureOff "Navigates to SIMATIC PLC system diagnostics for HMI_1"
      on Release: ActivateScreen("SIMATIC PLC system diagnostics", 0)
   Button "HmiScreenItemData_5" at 722,371 size 71x47; TextOn 'Online'; TextOff 'Set time'
      on Click: SetBit("write_time")
      on Release: ResetBit("write_time")
   IOField "I/O field_1" at 7,387 size 230x30; FormatPattern 9999999999999999999999999999999999999999
      ProcessValue <- "db_time_sync_time_local_READ"
   TextField "Text field_1" at 69,359 size 106x23; Text 'System time'
   TextField "Text field_2" at 317,360 size 89x23; Text 'Local time'
   IOField "I/O field_2" at 247,388 size 230x30; FormatPattern 9999999999999999999999999999999999999999
      ProcessValue <- "db_time_sync_time_system_READ"
   IOField "I/O field_3" at 486,388 size 230x30; FormatPattern 9999999999999999999999999999999999999999
      ProcessValue <- "db_time_sync_time_system_WRITE"
   TextField "Text field_4" at 564,360 size 74x23; Text 'Set time'

screen "Test" 800x480, template "Template_1"
   on GenerateScreen: SetTag("Tag_ScreenNumber", 5)
   Button "HmiScreenItemData_1" at 16,148 size 150x50; TextOn 'SIMATIC PLC system diagnostics'; TextOff 'Sello horizontal'; PictureOn "Navigates to SIMATIC PLC system diagnostics for HMI_1"; PictureOff "Navigates to SIMATIC PLC system diagnostics for HMI_1"
      on Release: ResetBit("Testhorizontalsealer_hmi")
      on Press: SetBit("Testhorizontalsealer_hmi")
      Appearance <- "Testhorizontalsealer_hmi"
   Button "HmiScreenItemData_2" at 16,260 size 150x50; TextOn 'SIMATIC PLC system diagnostics'; TextOff 'Cuchilla'; PictureOn "Navigates to SIMATIC PLC system diagnostics for HMI_1"; PictureOff "Navigates to SIMATIC PLC system diagnostics for HMI_1"
      on Release: ResetBit("TestKnife_hmi")
      on Press: SetBit("TestKnife_hmi")
      Appearance <- "TestKnife_hmi"
   Button "HmiScreenItemData_3" at 16,204 size 150x50; TextOn 'SIMATIC PLC system diagnostics'; TextOff 'Sello vertical'; PictureOn "Navigates to SIMATIC PLC system diagnostics for HMI_1"; PictureOff "Navigates to SIMATIC PLC system diagnostics for HMI_1"
      on Release: ResetBit("TestVerticalsealer_hmi")
      on Press: SetBit("TestVerticalsealer_hmi")
      Appearance <- "TestVerticalsealer_hmi"
   Button "HmiScreenItemData_4" at 16,92 size 150x50; TextOn 'SIMATIC PLC system diagnostics'; TextOff 'Codificador'; PictureOn "Navigates to SIMATIC PLC system diagnostics for HMI_1"; PictureOff "Navigates to SIMATIC PLC system diagnostics for HMI_1"
      on Release: ResetBit("Testdater_hmi")
      on Press: SetBit("Testdater_hmi")
      Appearance <- "Testdater_hmi"
   Button "HmiScreenItemData_5" at 220,260 size 150x50; TextOn 'SIMATIC PLC system diagnostics'; TextOff 'Banda arrastre'; PictureOn "Navigates to SIMATIC PLC system diagnostics for HMI_1"; PictureOff "Navigates to SIMATIC PLC system diagnostics for HMI_1"
      on Release: ResetBit("TestPuller_hmi")
      on Press: SetBit("TestPuller_hmi")
      Appearance <- "TestPuller_hmi"
   Button "HmiScreenItemData_6" at 219,92 size 150x50; TextOn 'SIMATIC PLC system diagnostics'; TextOff 'Dosificador'; PictureOn "Navigates to SIMATIC PLC system diagnostics for HMI_1"; PictureOff "Navigates to SIMATIC PLC system diagnostics for HMI_1"
      on Release: ResetBit("Testdoser_hmi")
      on Press: SetBit("Testdoser_hmi")
      Appearance <- "Testdoser_hmi"
   TextField "Text field_3" at 45,65 size 125x23; Text 'Accionamiento'
   Button "HmiScreenItemData_12" at 220,316 size 150x50; TextOn 'SIMATIC PLC system diagnostics'; TextOff 'Producto'; PictureOn "Navigates to SIMATIC PLC system diagnostics for HMI_1"; PictureOff "Navigates to SIMATIC PLC system diagnostics for HMI_1"
      on Release: ResetBit("TestFeeder_hmi")
      on Press: SetBit("TestFeeder_hmi")
      Appearance <- "TestFeeder_hmi"
   Button "HmiScreenItemData_13" at 219,148 size 150x50; TextOn 'SIMATIC PLC system diagnostics'; TextOff 'Agitador'; PictureOn "Navigates to SIMATIC PLC system diagnostics for HMI_1"; PictureOff "Navigates to SIMATIC PLC system diagnostics for HMI_1"
      on Release: ResetBit("TestBlender_hmi")
      on Press: SetBit("TestBlender_hmi")
      Appearance <- "TestBlender_hmi"
   Button "HmiScreenItemData_15" at 219,204 size 150x50; TextOn 'SIMATIC PLC system diagnostics'; TextOff 'Colector'; PictureOn "Navigates to SIMATIC PLC system diagnostics for HMI_1"; PictureOff "Navigates to SIMATIC PLC system diagnostics for HMI_1"
      on Release: ResetBit("TestCollector_hmi")
      on Press: SetBit("TestCollector_hmi")
      Appearance <- "TestCollector_hmi"

screen "SIMATIC PLC system diagnostics" 800x480, template "Template_1"
   on GenerateScreen: SetTag("Tag_ScreenNumber", 7)
   SysDiagControl "HmiScreenItemData" at 1,100 size 796x321

screen "User administration" 800x480, template "Template_1"
   on GenerateScreen: SetTag("Tag_ScreenNumber", 8)
   UserView "HmiScreenItemData" at 1,100 size 796x321
*)